// TwinCAT 3 PLC project IntelligenteWZM_PLCProject
// ProgramVersion: 3.1.4022.4
// libraries:
//   Tc2_Standard, * (Beckhoff Automation GmbH)
//   Tc2_System, * (Beckhoff Automation GmbH)
//   Tc3_Module, * (Beckhoff Automation GmbH)
//   VisuDialogs, * (System)
//   VisuSymbols,3.5.10.0,System
// project tree:
//   DUTs/ DW_TO_REAL.TcDUT
//   / GlobalTextList.TcGTLO (not stored), PlcTask.TcTTO, Visualization Manager.TcVMO (not stored)
//   GVLs/ GVarL.TcGVL
//   POUs/ ADAS_Kom.TcPOU, ANALOG_INPUT_EL3104.TcPOU, ANALOG_OUTPUT_EL4134.TcPOU (not stored), DATAMODULE.TcPOU (not stored), DATA_PREPARATION.TcPOU (not stored), DEFLECTION_CONTROL_FEED.TcPOU, DEFLECTION_CONTROL_POSITION.TcPOU (not stored), DP_CONFIG_IN_EL6731.TcPOU (not stored), DP_CONFIG_OUT_EL6731.TcPOU, ELLIP_FILTER.TcPOU (not stored), FORCE_SIGNALS.TcPOU, MAIN.TcPOU, MEAS_STIFFNESS_COLLISION.TcPOU (not stored), MEAS_STIFFNESS_PROCESS.TcPOU (not stored), Test.TcPOU (not stored), TOUCH_PROBE_LINE.TcPOU, VARIABLES.TcGVL (not stored), SENSOR_CONTROL_EL6751.TcPOU, SENSOR_SIGNALS_EL6751.TcPOU
//   VISUs/ Datamodule.TcVIS (not stored), PICTURES.TcIPO (not stored), VISUALISATION_DEFLEC_CONTROL.TcVIS, VISUALISATION_EMO2017.TcVIS, VISUALISATION_SENSOR_CONTROL.TcVIS, VISUALISATION_STIFFNESS_COLLISION.TcVIS, VISUALISATION_STIFFNESS_PROCESS.TcVIS (not stored)
// real-time tasks:
//   TASK PlcTask: cycle T#1ms, priority 20, ADS port 350
//   TASK Task 1: cycle T#10ms, priority 1, ADS port 301
// I/O:
//   DEVICE Device 2 (EtherCAT), AmsNetId 169.254.30.239.3.1
//     Term 1 (EK1100) [EK1100 EtherCAT Coupler (2A E-Bus)]
//       Term 2 (EL4134) [EL4134 4Ch. Ana. Output -10/+10V, 16bit]
//       Term 3 (EL3104) [EL3104 4Ch. Ana. Input +/-10V Diff.]
//       Term 4 (EL6731-0010) [EL6731-0010 PROFIBUS DP Slave]
//       Term 5 (EL6751) [EL6751 CANopen Master]
//       Term 6 (EL9512) [EL9512 Power supply terminal 12V]
//       Term 11 (EL9011) [EL9011 End Terminal]
//     Term 7 (EK1100) [EK1100 EtherCAT Coupler (2A E-Bus)]
//       Term 8 (EL3632) [EL3632 2Ch. IEPE Sensor]
//       Term 9 (EL3632) [EL3632 2Ch. IEPE Sensor]
//       Term 10 (EL3632) [EL3632 2Ch. IEPE Sensor]
//       Term 12 (EL9011) [EL9011 End Terminal]
//   DEVICE Device 1 (EL6731-0010), AmsNetId 169.254.30.239.2.1
//     PROFIBUS-Sinumerik (EL6731-0010) // Vendor: BECKHOFF Revision: Revision 2.00
//   DEVICE Device 3 (EL6751), AmsNetId 169.254.30.239.4.1
//     CAN-Sensors (CANopen Node)
// variable links:
//   IntelligenteWZM_PLCProject/IntelligenteWZM_PLCProject Instance <-> Device 1 (EL6731-0010)/PROFIBUS-Sinumerik (EL6731-0010)
//     PlcTask Inputs/VARIABLES.DP_MOSI_WORD_{1..4} <-> Module {5..8} (1 WORD Slave-In/Master-Out)/Inputs/1 WORD Slave-In/Master-Out_0_0  (4 links)
//     PlcTask Outputs/VARIABLES.DP_MISO_WORD_{1..4} <-> Module {1..4} (1 WORD Slave-Out/Master-In)/Outputs/1 WORD Slave-Out/Master-In_1_0  (4 links)
//   IntelligenteWZM_PLCProject/IntelligenteWZM_PLCProject Instance <-> Device 2 (EtherCAT)/Term 7 (EK1100)/Term 10 (EL3632)
//     PlcTask Inputs/VARIABLES.A_OVERSAMPLING_INPUT_5[0] <-> Ch1 Sample 0/Ch1 Value
//     PlcTask Inputs/VARIABLES.A_OVERSAMPLING_INPUT_5[1] <-> Ch1 Sample 1/Ch1 Value
//     PlcTask Inputs/VARIABLES.A_OVERSAMPLING_INPUT_5[2] <-> Ch1 Sample 2/Ch1 Value
//     PlcTask Inputs/VARIABLES.A_OVERSAMPLING_INPUT_5[3] <-> Ch1 Sample 3/Ch1 Value
//     PlcTask Inputs/VARIABLES.A_OVERSAMPLING_INPUT_5[4] <-> Ch1 Sample 4/Ch1 Value
//     PlcTask Inputs/VARIABLES.A_OVERSAMPLING_INPUT_5[5] <-> Ch1 Sample 5/Ch1 Value
//     PlcTask Inputs/VARIABLES.A_OVERSAMPLING_INPUT_5[6] <-> Ch1 Sample 6/Ch1 Value
//     PlcTask Inputs/VARIABLES.A_OVERSAMPLING_INPUT_5[7] <-> Ch1 Sample 7/Ch1 Value
//     PlcTask Inputs/VARIABLES.A_OVERSAMPLING_INPUT_5[8] <-> Ch1 Sample 8/Ch1 Value
//     PlcTask Inputs/VARIABLES.A_OVERSAMPLING_INPUT_5[9] <-> Ch1 Sample 9/Ch1 Value
//     PlcTask Inputs/VARIABLES.A_OVERSAMPLING_INPUT_6[0] <-> Ch2 Sample 0/Ch2 Value
//     PlcTask Inputs/VARIABLES.A_OVERSAMPLING_INPUT_6[1] <-> Ch2 Sample 1/Ch2 Value
//     PlcTask Inputs/VARIABLES.A_OVERSAMPLING_INPUT_6[2] <-> Ch2 Sample 2/Ch2 Value
//     PlcTask Inputs/VARIABLES.A_OVERSAMPLING_INPUT_6[3] <-> Ch2 Sample 3/Ch2 Value
//     PlcTask Inputs/VARIABLES.A_OVERSAMPLING_INPUT_6[4] <-> Ch2 Sample 4/Ch2 Value
//     PlcTask Inputs/VARIABLES.A_OVERSAMPLING_INPUT_6[5] <-> Ch2 Sample 5/Ch2 Value
//     PlcTask Inputs/VARIABLES.A_OVERSAMPLING_INPUT_6[6] <-> Ch2 Sample 6/Ch2 Value
//     PlcTask Inputs/VARIABLES.A_OVERSAMPLING_INPUT_6[7] <-> Ch2 Sample 7/Ch2 Value
//     PlcTask Inputs/VARIABLES.A_OVERSAMPLING_INPUT_6[8] <-> Ch2 Sample 8/Ch2 Value
//     PlcTask Inputs/VARIABLES.A_OVERSAMPLING_INPUT_6[9] <-> Ch2 Sample 9/Ch2 Value
//   IntelligenteWZM_PLCProject/IntelligenteWZM_PLCProject Instance <-> Device 2 (EtherCAT)/Term 7 (EK1100)/Term 8 (EL3632)
//     PlcTask Inputs/VARIABLES.A_OVERSAMPLING_INPUT_1[0] <-> Ch1 Sample 0/Ch1 Value
//     PlcTask Inputs/VARIABLES.A_OVERSAMPLING_INPUT_1[1] <-> Ch1 Sample 1/Ch1 Value
//     PlcTask Inputs/VARIABLES.A_OVERSAMPLING_INPUT_1[2] <-> Ch1 Sample 2/Ch1 Value
//     PlcTask Inputs/VARIABLES.A_OVERSAMPLING_INPUT_1[3] <-> Ch1 Sample 3/Ch1 Value
//     PlcTask Inputs/VARIABLES.A_OVERSAMPLING_INPUT_1[4] <-> Ch1 Sample 4/Ch1 Value
//     PlcTask Inputs/VARIABLES.A_OVERSAMPLING_INPUT_1[5] <-> Ch1 Sample 5/Ch1 Value
//     PlcTask Inputs/VARIABLES.A_OVERSAMPLING_INPUT_1[6] <-> Ch1 Sample 6/Ch1 Value
//     PlcTask Inputs/VARIABLES.A_OVERSAMPLING_INPUT_1[7] <-> Ch1 Sample 7/Ch1 Value
//     PlcTask Inputs/VARIABLES.A_OVERSAMPLING_INPUT_1[8] <-> Ch1 Sample 8/Ch1 Value
//     PlcTask Inputs/VARIABLES.A_OVERSAMPLING_INPUT_1[9] <-> Ch1 Sample 9/Ch1 Value
//     PlcTask Inputs/VARIABLES.A_OVERSAMPLING_INPUT_2[0] <-> Ch2 Sample 0/Ch2 Value
//     PlcTask Inputs/VARIABLES.A_OVERSAMPLING_INPUT_2[1] <-> Ch2 Sample 1/Ch2 Value
//     PlcTask Inputs/VARIABLES.A_OVERSAMPLING_INPUT_2[2] <-> Ch2 Sample 2/Ch2 Value
//     PlcTask Inputs/VARIABLES.A_OVERSAMPLING_INPUT_2[3] <-> Ch2 Sample 3/Ch2 Value
//     PlcTask Inputs/VARIABLES.A_OVERSAMPLING_INPUT_2[4] <-> Ch2 Sample 4/Ch2 Value
//     PlcTask Inputs/VARIABLES.A_OVERSAMPLING_INPUT_2[5] <-> Ch2 Sample 5/Ch2 Value
//     PlcTask Inputs/VARIABLES.A_OVERSAMPLING_INPUT_2[6] <-> Ch2 Sample 6/Ch2 Value
//     PlcTask Inputs/VARIABLES.A_OVERSAMPLING_INPUT_2[7] <-> Ch2 Sample 7/Ch2 Value
//     PlcTask Inputs/VARIABLES.A_OVERSAMPLING_INPUT_2[8] <-> Ch2 Sample 8/Ch2 Value
//     PlcTask Inputs/VARIABLES.A_OVERSAMPLING_INPUT_2[9] <-> Ch2 Sample 9/Ch2 Value
//   IntelligenteWZM_PLCProject/IntelligenteWZM_PLCProject Instance <-> Device 2 (EtherCAT)/Term 7 (EK1100)/Term 9 (EL3632)
//     PlcTask Inputs/VARIABLES.A_OVERSAMPLING_INPUT_3[0] <-> Ch1 Sample 0/Ch1 Value
//     PlcTask Inputs/VARIABLES.A_OVERSAMPLING_INPUT_3[1] <-> Ch1 Sample 1/Ch1 Value
//     PlcTask Inputs/VARIABLES.A_OVERSAMPLING_INPUT_3[2] <-> Ch1 Sample 2/Ch1 Value
//     PlcTask Inputs/VARIABLES.A_OVERSAMPLING_INPUT_3[3] <-> Ch1 Sample 3/Ch1 Value
//     PlcTask Inputs/VARIABLES.A_OVERSAMPLING_INPUT_3[4] <-> Ch1 Sample 4/Ch1 Value
//     PlcTask Inputs/VARIABLES.A_OVERSAMPLING_INPUT_3[5] <-> Ch1 Sample 5/Ch1 Value
//     PlcTask Inputs/VARIABLES.A_OVERSAMPLING_INPUT_3[6] <-> Ch1 Sample 6/Ch1 Value
//     PlcTask Inputs/VARIABLES.A_OVERSAMPLING_INPUT_3[7] <-> Ch1 Sample 7/Ch1 Value
//     PlcTask Inputs/VARIABLES.A_OVERSAMPLING_INPUT_3[8] <-> Ch1 Sample 8/Ch1 Value
//     PlcTask Inputs/VARIABLES.A_OVERSAMPLING_INPUT_3[9] <-> Ch1 Sample 9/Ch1 Value
//     PlcTask Inputs/VARIABLES.A_OVERSAMPLING_INPUT_4[0] <-> Ch2 Sample 0/Ch2 Value
//     PlcTask Inputs/VARIABLES.A_OVERSAMPLING_INPUT_4[1] <-> Ch2 Sample 1/Ch2 Value
//     PlcTask Inputs/VARIABLES.A_OVERSAMPLING_INPUT_4[2] <-> Ch2 Sample 2/Ch2 Value
//     PlcTask Inputs/VARIABLES.A_OVERSAMPLING_INPUT_4[3] <-> Ch2 Sample 3/Ch2 Value
//     PlcTask Inputs/VARIABLES.A_OVERSAMPLING_INPUT_4[4] <-> Ch2 Sample 4/Ch2 Value
//     PlcTask Inputs/VARIABLES.A_OVERSAMPLING_INPUT_4[5] <-> Ch2 Sample 5/Ch2 Value
//     PlcTask Inputs/VARIABLES.A_OVERSAMPLING_INPUT_4[6] <-> Ch2 Sample 6/Ch2 Value
//     PlcTask Inputs/VARIABLES.A_OVERSAMPLING_INPUT_4[7] <-> Ch2 Sample 7/Ch2 Value
//     PlcTask Inputs/VARIABLES.A_OVERSAMPLING_INPUT_4[8] <-> Ch2 Sample 8/Ch2 Value
//     PlcTask Inputs/VARIABLES.A_OVERSAMPLING_INPUT_4[9] <-> Ch2 Sample 9/Ch2 Value
//   IntelligenteWZM_PLCProject/IntelligenteWZM_PLCProject Instance <-> Device 3 (EL6751)/CAN-Sensors (CANopen Node)
//     PlcTask Inputs/VARIABLES.CAN_SENSOR_{1..10} <-> Sensor ID {1..10}/Inputs/CAN_IN_MESSAGE_D{1..10}  (10 links)
//     PlcTask Outputs/VARIABLES.CAN_HUB <-> HUB Control ID 0/Outputs/CAN_OUT_MESSAGE_CONTROL

CONFIGURATION IntelligenteWZM_PLCProject
    RESOURCE PLC ON TwinCAT3
        TASK PlcTask(INTERVAL := T#1ms, PRIORITY := 20);
        PROGRAM MAIN WITH PlcTask : MAIN;
    END_RESOURCE
END_CONFIGURATION

// ---- DUTs/DW_TO_REAL.TcDUT
TYPE DW_TO_REAL :
UNION
	IntAsWord : ARRAY[0..1] OF WORD;
	IntAsReal: REAL;
END_UNION
END_TYPE

// ---- GVLs/GVarL.TcGVL
VAR_GLOBAL
	///ADAS 
	iSignalID: ARRAY[0..20] OF BYTE;
	iAchseID: ARRAY[0..20] OF BYTE;
	iComCylce: BYTE := 20;
	iMode: INT := 10;
	iTracks: UINT;
	///Position x
	X_Machine_CS AT %Q*: LREAL;
	///Position y
	Y_Machine_CS AT %Q*: LREAL;
	///Position z
	Z_Machine_CS AT %Q*: LREAL;
	///Position c
	C_Machine_CS AT %Q*: LREAL;
	///Position b
	B_Machine_CS AT %Q*: LREAL;
	///Soll-Position x
	X_Machine_CS_soll AT %Q*: LREAL;
	///Geschwindigkeit x
	X_V_Machine_CS AT %Q*: LREAL;
	///Geschwindigkeit y
	Y_V_Machine_CS AT %Q*: LREAL;
	///Geschwindigkeit z
	Z_V_Machine_CS AT %Q*: LREAL;
	///Geschwindigkeit c
	C_V_Machine_CS AT %Q*: LREAL;
	///Geschwindigkeit b
	B_V_Machine_CS AT %Q*: LREAL;
	///Drehzahl n
	n_Spindle AT %Q*: LREAL;
	///Beschleunigung x
	X_a_Machine_CS AT %Q*: LREAL;
	///Beschleunigung y
	Y_a_Machine_CS AT %Q*: LREAL;
	///Beschleunigung z
	Z_a_Machine_CS AT %Q*: LREAL;
	///Beschleunigung c
	C_a_Machine_CS AT %Q*: LREAL;
	///Beschleunigung b
	B_a_Machine_CS AT %Q*: LREAL;
	///Strom x
	X_I AT %Q*: LREAL;
	///Strom y
	Y_I AT %Q*: LREAL;
	///Strom z
	Z_I AT %Q*: LREAL;
	///Strom c
	C_I AT %Q*: LREAL;
	///Strom b
	B_I AT %Q*: LREAL;
	///Strom Spindel
	n_I AT %Q*: LREAL;
	Data: uCCDatagram;
	///CCDataStreamSetupOUT 	 		:sCCDataStreamSetup;
	CCDataStreamSetupOUT AT %Q*: sCCDataStreamSetup;
	bGO: BOOL;

	XSynVar: LREAL;
END_VAR

VAR_GLOBAL CONSTANT
	///ADAS
	gVar_NumberOfAdasTracks: INT := 30;
END_VAR

// ---- POUs/MAIN.TcPOU
PROGRAM MAIN
VAR_INPUT
//ADAS
	ADAS_in		AT %I* 	: ARRAY[0..63] OF WORD; //ADAS_Rohdaten
END_VAR


IF FORCE_RESET=1 THEN
	RESULT[0]:=0;
	PTS_MEASUREMENT_HISTOGRAM_2[2]:=0;
	RESULT[1]:=0;
END_IF

IF VarTest = TRUE THEN
	VarTest := FALSE;
END_IF

IF VarTest = FALSE THEN
	VarTest := TRUE;
END_IF

ANALOG_INPUT_EL3104();
//ANALOG_OUTPUT_EL4134();
DP_CONFIG_IN_EL6731();
SENSOR_CONTROL_EL6751();
SENSOR_SIGNALS_EL6751();
FORCE_SIGNALS();
//Test();
DATAMODULE();

MEAS_STIFFNESS_COLLISION();
MEAS_STIFFNESS_PROCESS();
DEFLECTION_CONTROL_FEED();
DEFLECTION_CONTROL_POSITION();
TOUCH_PROBE_LINE();
DP_CONFIG_OUT_EL6731();


//ADAS Daten
	//x-Achse (soll alles stimmen)
X_Machine_CS 		:= DINT_TO_LREAL(ADAS_Kom.adasData[1])	/ 10000; //Umrechnung in: mm -> /10000 (10000 inkremente sind 1mm)
X_Machine_CS_soll 	:= DINT_TO_LREAL(ADAS_Kom.adasData[27])	/ 10000; //Umrechnung in: mm -> /10000 (10000 inkremente sind 1mm)
X_V_Machine_CS 		:= DINT_TO_LREAL(ADAS_Kom.adasData[6])	/ 10000; //Umrechnung in: mm/s-> /10000
X_a_Machine_CS 		:= DINT_TO_LREAL(ADAS_Kom.adasData[12])	/ 10000; //Umrechnung in: mm/s²-> /10000
X_I					:= DINT_TO_LREAL(ADAS_Kom.adasData[18])	/ 1000;  //Umrechnung in: A -> /1000

	//y-Achse  (soll alles stimmen)
Y_Machine_CS 		:= DINT_TO_LREAL(ADAS_Kom.adasData[2]) 	/ 10000; //Umrechnung in: mm -> /10000
Y_V_Machine_CS 		:= DINT_TO_LREAL(ADAS_Kom.adasData[7]) 	/ 10000; //Umrechnung in: mm/s-> /10000
Y_a_Machine_CS 		:= DINT_TO_LREAL(ADAS_Kom.adasData[13])	/ 10000; //Umrechnung in: mm/s²-> /10000
Y_I					:= DINT_TO_LREAL(ADAS_Kom.adasData[19])	/ 1000;  //Umrechnung in: A -> /1000
	//z-Achse (soll alles stimmen)
Z_Machine_CS 		:= DINT_TO_LREAL(ADAS_Kom.adasData[3]) 	/ 10000; //Umrechnung in: mm -> /10000
Z_V_Machine_CS 		:= DINT_TO_LREAL(ADAS_Kom.adasData[8]) 	/ 10000; //Umrechnung in: mm/s-> /10000
Z_a_Machine_CS 		:= DINT_TO_LREAL(ADAS_Kom.adasData[14])	/ 10000; //Umrechnung in: mm/s²-> /10000
Z_I					:= DINT_TO_LREAL(ADAS_Kom.adasData[20])	/ 1000;  //Umrechnung in: A -> /1000
	//C-Achse (soll alles stimmen)
C_Machine_CS 		:= DINT_TO_LREAL(ADAS_Kom.adasData[4]) 	/ 10000; //Umrechnung in: mm -> /10000
C_V_Machine_CS 		:= DINT_TO_LREAL(ADAS_Kom.adasData[9]) 	/ 10000; //Umrechnung in: mm/s-> /10000
C_a_Machine_CS 		:= DINT_TO_LREAL(ADAS_Kom.adasData[15])	/ 10000; //Umrechnung in: mm/s²-> /10000
C_I 				:= DINT_TO_LREAL(ADAS_Kom.adasData[21])	/ 1000;  //Umrechnung in: A -> /1000
	//B-Achse (B_Machine_CS wid von Spinel beschrieben)
B_Machine_CS		:= DINT_TO_LREAL(ADAS_Kom.adasData[24]) / 10000; //Umrechnung in: mm -> /10000 //b
B_V_Machine_CS 		:= DINT_TO_LREAL(ADAS_Kom.adasData[10]) / 10000; //Umrechnung in: mm/s-> /10000
B_a_Machine_CS 		:= DINT_TO_LREAL(ADAS_Kom.adasData[16]) / 10000; //Umrechnung in: mm/s²-> /10000
B_I 				:= DINT_TO_LREAL(ADAS_Kom.adasData[22]) / 1000;  //Umrechnung in: A -> /1000
	//Spindel
n_Spindle 			:= (DINT_TO_LREAL(ADAS_Kom.adasData[5])/360)*60/10000 ; //kommt in milli°/s Umrechnung in: 1/min-> *0,166667
n_I 				:= DINT_TO_LREAL(ADAS_Kom.adasData[25])/1000; //Umrechnung in: A -> /1000

END_PROGRAM

// ---- POUs/ANALOG_INPUT_EL3104.TcPOU
PROGRAM ANALOG_INPUT_EL3104
VAR
END_VAR


A_SIGNAL_1 := INT_TO_REAL(A_INPUT_1)*A_GAIN_1*10/ 32767;
A_SIGNAL_2 := INT_TO_REAL(A_INPUT_2)*A_GAIN_2*10/ 32767;
A_SIGNAL_3 := INT_TO_REAL(A_INPUT_3)*A_GAIN_3*10/ 32767;
A_SIGNAL_4 := INT_TO_REAL(A_INPUT_4)*A_GAIN_4*10/ 32767;

END_PROGRAM

// ---- POUs/SENSOR_CONTROL_EL6751.TcPOU
PROGRAM SENSOR_CONTROL_EL6751
VAR
	Samp: WORD:=0;	
	FigArray: ARRAY [0..7] OF USINT :=[0, 0, 0, 0, 0, 0, 0, 0];
	Previous: USINT:=16#0;
END_VAR

HUB_STATE:=FALSE; 

IF CAN_TRIGGER_STATE=1 AND M_PER_FRAME=1 THEN
	CAN_CONTROL_FRAME:=FigArray;
	IF samp>K_Trigger THEN			// Can occurs by changing M_PER_FRAME from 2,3 or 4 to 1 
		samp:=0;
	END_IF
	Samp:=Samp+1;
	IF Samp=K_Trigger THEN
		CAN_CONTROL_FRAME[0]:=16#3;
		CAN_CONTROL_FRAME[2]:=16#1;
		CAN_CONTROL_FRAME[4]:=N_SAMPLES_PER_M;
		CASE Previous OF
			16#0: 	CAN_CONTROL_FRAME[3]:=16#0;
					Previous:=16#1;
			16#1: 	CAN_CONTROL_FRAME[3]:=16#1;
					Previous:=16#0;
		END_CASE
		SIGNAL_SYNCH:=1;
		Samp:=0;
		CAN_HUB:=CAN_CONTROL_FRAME;	
	END_IF	
	HUB_STATE:=TRUE;
END_IF



IF CAN_TRIGGER_STATE=1 AND M_PER_FRAME=2 THEN
	CAN_CONTROL_FRAME:=FigArray;
	Samp:=Samp+1;
	IF Samp=K_Trigger OR Samp=(2*K_Trigger) THEN
		CAN_CONTROL_FRAME[0]:=16#3;
		CAN_CONTROL_FRAME[2]:=16#2;
		CAN_CONTROL_FRAME[4]:=N_SAMPLES_PER_M;
		IF Samp=K_Trigger THEN
			CAN_CONTROL_FRAME[3]:=16#1;
			SIGNAL_SYNCH:=1;
		END_IF
		IF Samp=(2*K_Trigger) THEN
			CAN_CONTROL_FRAME[3]:=16#2;
			SIGNAL_SYNCH:=2;
			Samp:=0;
		END_IF
		CAN_HUB:=CAN_CONTROL_FRAME;	
	END_IF
	HUB_STATE:=TRUE;
END_IF



IF CAN_TRIGGER_STATE=1 AND M_PER_FRAME=3 THEN
	CAN_CONTROL_FRAME:=FigArray;
	Samp:=Samp+1;
	IF Samp=K_Trigger OR Samp=(2*K_Trigger) OR Samp=(3*K_Trigger) THEN
		CAN_CONTROL_FRAME[0]:=16#3;
		CAN_CONTROL_FRAME[2]:=16#3;
		CAN_CONTROL_FRAME[4]:=N_SAMPLES_PER_M;
		IF Samp=K_Trigger THEN
			CAN_CONTROL_FRAME[3]:=16#1;
			SIGNAL_SYNCH:=1;
		END_IF
		IF Samp=(2*K_Trigger) THEN
			CAN_CONTROL_FRAME[3]:=16#2;
			SIGNAL_SYNCH:=2;
		END_IF
		IF Samp=(3*K_Trigger) THEN
			CAN_CONTROL_FRAME[3]:=16#3;
			SIGNAL_SYNCH:=3;
			Samp:=0;
		END_IF
		CAN_HUB:=CAN_CONTROL_FRAME;	
	END_IF
	HUB_STATE:=TRUE;
END_IF


IF CAN_TRIGGER_STATE=1 AND M_PER_FRAME=4 THEN
	CAN_CONTROL_FRAME:=FigArray;
	Samp:=Samp+1;
	IF Samp=K_Trigger OR Samp=(2*K_Trigger) OR Samp=(3*K_Trigger) OR Samp=(4*K_Trigger)  THEN
		CAN_CONTROL_FRAME[0]:=16#3;
		CAN_CONTROL_FRAME[2]:=16#4;
		CAN_CONTROL_FRAME[4]:=N_SAMPLES_PER_M;
		IF Samp=K_Trigger THEN
			CAN_CONTROL_FRAME[3]:=16#1;
			SIGNAL_SYNCH:=1;
		END_IF
		IF Samp=(2*K_Trigger) THEN
			CAN_CONTROL_FRAME[3]:=16#2;
			SIGNAL_SYNCH:=2;
		END_IF
		IF Samp=(3*K_Trigger) THEN
			CAN_CONTROL_FRAME[3]:=16#3;
			SIGNAL_SYNCH:=3;
		END_IF
		IF Samp=(4*K_Trigger) THEN
			CAN_CONTROL_FRAME[3]:=16#4;
			SIGNAL_SYNCH:=4;
			Samp:=0;
		END_IF
		CAN_HUB:=CAN_CONTROL_FRAME;		
	END_IF
	HUB_STATE:=TRUE;
END_IF

IF CAN_CONTROL_STATE=0 THEN
	CAN_CONTROL_FRAME:=FigArray;
	CAN_CONTROL_FRAME[0]:=16#0;
	CAN_HUB:=CAN_CONTROL_FRAME;
	CAN_CONTROL_STATE:=11;
	HUB_STATE:=TRUE;
END_IF

IF CAN_CONTROL_STATE=1 THEN
	CAN_CONTROL_FRAME:=FigArray;
	CAN_CONTROL_FRAME[0]:=16#1;
	CAN_HUB:=CAN_CONTROL_FRAME;
	CAN_CONTROL_STATE:=11;
	HUB_STATE:=TRUE;
END_IF

IF CAN_CONTROL_STATE=2 THEN
	CAN_CONTROL_FRAME:=FigArray;
	CAN_CONTROL_FRAME[0]:=16#2;
	CAN_HUB:=CAN_CONTROL_FRAME;
	CAN_CONTROL_STATE:=11;
	HUB_STATE:=TRUE;
END_IF

IF CAN_CONTROL_STATE=3 THEN
	CAN_CONTROL_FRAME:=CAN_PARAMETER_FRAME;
	CAN_HUB:=CAN_CONTROL_FRAME;
	CAN_CONTROL_STATE:=11;
	CAN_PARAMETER_FRAME:=FigArray;
	HUB_STATE:=TRUE;
END_IF

END_PROGRAM

// ---- POUs/SENSOR_SIGNALS_EL6751.TcPOU
PROGRAM SENSOR_SIGNALS_EL6751
VAR
	FILTER_S1:ELLIP_FILTER;
	FILTER_S2:ELLIP_FILTER;
	FILTER_S3:ELLIP_FILTER;
	FILTER_S4:ELLIP_FILTER;
	FILTER_S5:ELLIP_FILTER;
	FILTER_S6:ELLIP_FILTER;
	FILTER_S7:ELLIP_FILTER;
	FILTER_S8:ELLIP_FILTER;
	FILTER_S9:ELLIP_FILTER;
	FILTER_S10:ELLIP_FILTER;
	
	
	Calc_Dev: ARRAY[1..3,1..10] OF LREAL:=[0, 0, 0, 0, 0, 0, 0, 0, 0, 0, 0, 0, 0, 0, 0, 0, 0, 0, 0, 0, 0, 0, 0, 0, 0, 0, 0, 0, 0, 0 ];
	k: WORD;
	Signal_5: WORD:=0;
	Signal_1: WORD:=0;
	Mem_Signal_1: ARRAY[1..10] OF WORD:=[0,0,0,0,0,0,0,0,0,0];
	N_Mem_Sig_1: ARRAY[1..10] OF WORD:=[0,0,0,0,0,0,0,0,0,0];
	N_Dev: WORD:=500;
	
END_VAR

//SENSOR 1
SIGNAL_SENSOR_1[1]:=SHL(CAN_SENSOR_1[0],8)+CAN_SENSOR_1[1];
SIGNAL_SENSOR_1[2]:=SHL(CAN_SENSOR_1[2],8)+CAN_SENSOR_1[3];
SIGNAL_SENSOR_1[3]:=SHL(CAN_SENSOR_1[4],8)+CAN_SENSOR_1[5];
SIGNAL_SENSOR_1[4]:=SHL(CAN_SENSOR_1[6],8)+CAN_SENSOR_1[7];
CASE SIGNAL_SYNCH OF
	1: SIGNAL_SENSOR_1[5]:=SIGNAL_SENSOR_1[1];
	2: SIGNAL_SENSOR_1[5]:=SIGNAL_SENSOR_1[2];
	3: SIGNAL_SENSOR_1[5]:=SIGNAL_SENSOR_1[3];
	4: SIGNAL_SENSOR_1[5]:=SIGNAL_SENSOR_1[4];
END_CASE

//SENSOR 2
SIGNAL_SENSOR_2[1]:=SHL(CAN_SENSOR_2[0],8)+CAN_SENSOR_2[1];
SIGNAL_SENSOR_2[2]:=SHL(CAN_SENSOR_2[2],8)+CAN_SENSOR_2[3];
SIGNAL_SENSOR_2[3]:=SHL(CAN_SENSOR_2[4],8)+CAN_SENSOR_2[5];
SIGNAL_SENSOR_2[4]:=SHL(CAN_SENSOR_2[6],8)+CAN_SENSOR_2[7];
CASE SIGNAL_SYNCH OF
	1: SIGNAL_SENSOR_2[5]:=SIGNAL_SENSOR_2[1];
	2: SIGNAL_SENSOR_2[5]:=SIGNAL_SENSOR_2[2];
	3: SIGNAL_SENSOR_2[5]:=SIGNAL_SENSOR_2[3];
	4: SIGNAL_SENSOR_2[5]:=SIGNAL_SENSOR_2[4];
END_CASE

//SENSOR 3
SIGNAL_SENSOR_3[1]:=SHL(CAN_SENSOR_3[0],8)+CAN_SENSOR_3[1];
SIGNAL_SENSOR_3[2]:=SHL(CAN_SENSOR_3[2],8)+CAN_SENSOR_3[3];
SIGNAL_SENSOR_3[3]:=SHL(CAN_SENSOR_3[4],8)+CAN_SENSOR_3[5];
SIGNAL_SENSOR_3[4]:=SHL(CAN_SENSOR_3[6],8)+CAN_SENSOR_3[7];
CASE SIGNAL_SYNCH OF
	1: SIGNAL_SENSOR_3[5]:=SIGNAL_SENSOR_3[1];
	2: SIGNAL_SENSOR_3[5]:=SIGNAL_SENSOR_3[2];
	3: SIGNAL_SENSOR_3[5]:=SIGNAL_SENSOR_3[3];
	4: SIGNAL_SENSOR_3[5]:=SIGNAL_SENSOR_3[4];
END_CASE

//SENSOR 4
SIGNAL_SENSOR_4[1]:=SHL(CAN_SENSOR_4[0],8)+CAN_SENSOR_4[1];
SIGNAL_SENSOR_4[2]:=SHL(CAN_SENSOR_4[2],8)+CAN_SENSOR_4[3];
SIGNAL_SENSOR_4[3]:=SHL(CAN_SENSOR_4[4],8)+CAN_SENSOR_4[5];
SIGNAL_SENSOR_4[4]:=SHL(CAN_SENSOR_4[6],8)+CAN_SENSOR_4[7];
CASE SIGNAL_SYNCH OF
	1: SIGNAL_SENSOR_4[5]:=SIGNAL_SENSOR_4[1];
	2: SIGNAL_SENSOR_4[5]:=SIGNAL_SENSOR_4[2];
	3: SIGNAL_SENSOR_4[5]:=SIGNAL_SENSOR_4[3];
	4: SIGNAL_SENSOR_4[5]:=SIGNAL_SENSOR_4[4];
END_CASE

//SENSOR 5
SIGNAL_SENSOR_5[1]:=SHL(CAN_SENSOR_5[0],8)+CAN_SENSOR_5[1];
SIGNAL_SENSOR_5[2]:=SHL(CAN_SENSOR_5[2],8)+CAN_SENSOR_5[3];
SIGNAL_SENSOR_5[3]:=SHL(CAN_SENSOR_5[4],8)+CAN_SENSOR_5[5];
SIGNAL_SENSOR_5[4]:=SHL(CAN_SENSOR_5[6],8)+CAN_SENSOR_5[7];
CASE SIGNAL_SYNCH OF
	1: SIGNAL_SENSOR_5[5]:=SIGNAL_SENSOR_5[1];
	2: SIGNAL_SENSOR_5[5]:=SIGNAL_SENSOR_5[2];
	3: SIGNAL_SENSOR_5[5]:=SIGNAL_SENSOR_5[3];
	4: SIGNAL_SENSOR_5[5]:=SIGNAL_SENSOR_5[4];
END_CASE

//SENSOR 6
SIGNAL_SENSOR_6[1]:=SHL(CAN_SENSOR_6[0],8)+CAN_SENSOR_6[1];
SIGNAL_SENSOR_6[2]:=SHL(CAN_SENSOR_6[2],8)+CAN_SENSOR_6[3];
SIGNAL_SENSOR_6[3]:=SHL(CAN_SENSOR_6[4],8)+CAN_SENSOR_6[5];
SIGNAL_SENSOR_6[4]:=SHL(CAN_SENSOR_6[6],8)+CAN_SENSOR_6[7];
CASE SIGNAL_SYNCH OF
	1: SIGNAL_SENSOR_6[5]:=SIGNAL_SENSOR_6[1];
	2: SIGNAL_SENSOR_6[5]:=SIGNAL_SENSOR_6[2];
	3: SIGNAL_SENSOR_6[5]:=SIGNAL_SENSOR_6[3];
	4: SIGNAL_SENSOR_6[5]:=SIGNAL_SENSOR_6[4];
END_CASE

//SENSOR 7
SIGNAL_SENSOR_7[1]:=SHL(CAN_SENSOR_7[0],8)+CAN_SENSOR_7[1];
SIGNAL_SENSOR_7[2]:=SHL(CAN_SENSOR_7[2],8)+CAN_SENSOR_7[3];
SIGNAL_SENSOR_7[3]:=SHL(CAN_SENSOR_7[4],8)+CAN_SENSOR_7[5];
SIGNAL_SENSOR_7[4]:=SHL(CAN_SENSOR_7[6],8)+CAN_SENSOR_7[7];
CASE SIGNAL_SYNCH OF
	1: SIGNAL_SENSOR_7[5]:=SIGNAL_SENSOR_7[1];
	2: SIGNAL_SENSOR_7[5]:=SIGNAL_SENSOR_7[2];
	3: SIGNAL_SENSOR_7[5]:=SIGNAL_SENSOR_7[3];
	4: SIGNAL_SENSOR_7[5]:=SIGNAL_SENSOR_7[4];
END_CASE

//SENSOR 8
SIGNAL_SENSOR_8[1]:=SHL(CAN_SENSOR_8[0],8)+CAN_SENSOR_8[1];
SIGNAL_SENSOR_8[2]:=SHL(CAN_SENSOR_8[2],8)+CAN_SENSOR_8[3];
SIGNAL_SENSOR_8[3]:=SHL(CAN_SENSOR_8[4],8)+CAN_SENSOR_8[5];
SIGNAL_SENSOR_8[4]:=SHL(CAN_SENSOR_8[6],8)+CAN_SENSOR_8[7];
CASE SIGNAL_SYNCH OF
	1: SIGNAL_SENSOR_8[5]:=SIGNAL_SENSOR_8[1];
	2: SIGNAL_SENSOR_8[5]:=SIGNAL_SENSOR_8[2];
	3: SIGNAL_SENSOR_8[5]:=SIGNAL_SENSOR_8[3];
	4: SIGNAL_SENSOR_8[5]:=SIGNAL_SENSOR_8[4];
END_CASE

//SENSOR 9
SIGNAL_SENSOR_9[1]:=SHL(CAN_SENSOR_9[0],8)+CAN_SENSOR_9[1];
SIGNAL_SENSOR_9[2]:=SHL(CAN_SENSOR_9[2],8)+CAN_SENSOR_9[3];
SIGNAL_SENSOR_9[3]:=SHL(CAN_SENSOR_9[4],8)+CAN_SENSOR_9[5];
SIGNAL_SENSOR_9[4]:=SHL(CAN_SENSOR_9[6],8)+CAN_SENSOR_9[7];
CASE SIGNAL_SYNCH OF
	1: SIGNAL_SENSOR_9[5]:=SIGNAL_SENSOR_9[1];
	2: SIGNAL_SENSOR_9[5]:=SIGNAL_SENSOR_9[2];
	3: SIGNAL_SENSOR_9[5]:=SIGNAL_SENSOR_9[3];
	4: SIGNAL_SENSOR_9[5]:=SIGNAL_SENSOR_9[4];
END_CASE

//SENSOR 10
SIGNAL_SENSOR_10[1]:=SHL(CAN_SENSOR_10[0],8)+CAN_SENSOR_10[1];
SIGNAL_SENSOR_10[2]:=SHL(CAN_SENSOR_10[2],8)+CAN_SENSOR_10[3];
SIGNAL_SENSOR_10[3]:=SHL(CAN_SENSOR_10[4],8)+CAN_SENSOR_10[5];
SIGNAL_SENSOR_10[4]:=SHL(CAN_SENSOR_10[6],8)+CAN_SENSOR_10[7];
CASE SIGNAL_SYNCH OF
	1: SIGNAL_SENSOR_10[5]:=SIGNAL_SENSOR_10[1];
	2: SIGNAL_SENSOR_10[5]:=SIGNAL_SENSOR_10[2];
	3: SIGNAL_SENSOR_10[5]:=SIGNAL_SENSOR_10[3];
	4: SIGNAL_SENSOR_10[5]:=SIGNAL_SENSOR_10[4];
END_CASE

// SIGNAL FILTERING
FILTER_S1(ssMethodType:=1 , IN:= SIGNAL_SENSOR_1[5], OUT=> SIGNAL_SENSOR_1_FLT);
FILTER_S2(ssMethodType:=1 , IN:= SIGNAL_SENSOR_2[5], OUT=> SIGNAL_SENSOR_2_FLT);
FILTER_S3(ssMethodType:=1 , IN:= SIGNAL_SENSOR_3[5], OUT=> SIGNAL_SENSOR_3_FLT);
FILTER_S4(ssMethodType:=1 , IN:= SIGNAL_SENSOR_4[5], OUT=> SIGNAL_SENSOR_4_FLT);
FILTER_S5(ssMethodType:=1 , IN:= SIGNAL_SENSOR_5[5], OUT=> SIGNAL_SENSOR_5_FLT);
FILTER_S6(ssMethodType:=1 , IN:= SIGNAL_SENSOR_6[5], OUT=> SIGNAL_SENSOR_6_FLT);
FILTER_S7(ssMethodType:=1 , IN:= SIGNAL_SENSOR_7[5], OUT=> SIGNAL_SENSOR_7_FLT);
FILTER_S8(ssMethodType:=1 , IN:= SIGNAL_SENSOR_8[5], OUT=> SIGNAL_SENSOR_8_FLT);
FILTER_S9(ssMethodType:=1 , IN:= SIGNAL_SENSOR_9[5], OUT=> SIGNAL_SENSOR_9_FLT);
FILTER_S10(ssMethodType:=1 , IN:= SIGNAL_SENSOR_10[5], OUT=> SIGNAL_SENSOR_10_FLT);

// SIGNAL DEVIATION AND SIGNAL STATE
FOR k:=1 TO 10 BY 1 DO
	Calc_Dev[1,k]:=Calc_Dev[1,k]+1;
	CASE k OF
		1: 	Signal_5:=SIGNAL_SENSOR_1[5];
			Signal_1:=SIGNAL_SENSOR_1[1];
		2: 	Signal_5:=SIGNAL_SENSOR_2[5];
			Signal_1:=SIGNAL_SENSOR_2[1];
		3: 	Signal_5:=SIGNAL_SENSOR_3[5];
			Signal_1:=SIGNAL_SENSOR_3[1];
		4: 	Signal_5:=SIGNAL_SENSOR_4[5];
			Signal_1:=SIGNAL_SENSOR_4[1];
		5: 	Signal_5:=SIGNAL_SENSOR_5[5];
			Signal_1:=SIGNAL_SENSOR_5[1];
		6: 	Signal_5:=SIGNAL_SENSOR_6[5];
			Signal_1:=SIGNAL_SENSOR_6[1];
		7: 	Signal_5:=SIGNAL_SENSOR_7[5];
			Signal_1:=SIGNAL_SENSOR_7[1];
		8: 	Signal_5:=SIGNAL_SENSOR_8[5];
			Signal_1:=SIGNAL_SENSOR_8[1];
		9: 	Signal_5:=SIGNAL_SENSOR_9[5];
			Signal_1:=SIGNAL_SENSOR_9[1];
		10: Signal_5:=SIGNAL_SENSOR_10[5];
			Signal_1:=SIGNAL_SENSOR_10[1];	
	END_CASE
	
	IF Calc_Dev[1,k]<N_Dev THEN
		Calc_Dev[2,k]:=Calc_Dev[2,k]+EXPT(WORD_TO_LREAL(Signal_5),2)/(N_Dev-1);
		Calc_Dev[3,k]:=Calc_Dev[3,k]+WORD_TO_LREAL(Signal_5);
	END_IF
	
	IF Calc_Dev[1,k]=N_Dev THEN
		IF Calc_Dev[2,k]-(EXPT(Calc_Dev[3,k],2)/EXPT((N_Dev-1),2))>=0 THEN
			SIGNAL_DEVIATION[k]:=LREAL_TO_WORD(3*SQRT(Calc_Dev[2,k]-(EXPT(Calc_Dev[3,k],2)/EXPT((N_Dev-1),2))));
			Calc_Dev[1,k]:=0;
			Calc_Dev[2,k]:=0;
			Calc_Dev[3,k]:=0;
			ELSE
				Calc_Dev[1,k]:=0;
				Calc_Dev[2,k]:=0;
				Calc_Dev[3,k]:=0;
				SIGNAL_DEVIATION[k]:=0;
		END_IF
	END_IF
	
	IF Signal_1<>Mem_Signal_1[k] THEN
		N_Mem_Sig_1[k]:=0;
		Mem_Signal_1[k]:=Signal_1;
		ELSE
		N_Mem_Sig_1[k]:=N_Mem_Sig_1[k]+1;
		Mem_Signal_1[k]:=Signal_1;
	END_IF
	
	IF N_Mem_Sig_1[k]< N_Dev THEN
		SENSOR_STATE[k]:=1;
		ELSE
			SENSOR_STATE[k]:=0;	
			SIGNAL_DEVIATION[k]:=0;	
	END_IF
	
END_FOR

END_PROGRAM

// ---- POUs/FORCE_SIGNALS.TcPOU
PROGRAM FORCE_SIGNALS
VAR
	RESET_FORCE_VAL: ARRAY[1..3] OF REAL := [0,0,0];
	FORCE_ROW: ARRAY[1..3] OF REAL;
	FORCE_SUM: ARRAY[1..3] OF REAL:= [0,0,0];
	INK: INT:=0;
	
	FILTER_FX:ELLIP_FILTER;
	FILTER_FY:ELLIP_FILTER;
	FILTER_FZ:ELLIP_FILTER;
	
	
END_VAR

FORCE_ROW[1]:=(FC_MATRIX_X[1]*SIGNAL_SENSOR_1[1]+FC_MATRIX_X[2]*SIGNAL_SENSOR_2[1]+FC_MATRIX_X[3]*SIGNAL_SENSOR_3[1]+FC_MATRIX_X[4]*SIGNAL_SENSOR_4[1]+FC_MATRIX_X[5]*SIGNAL_SENSOR_5[1]+FC_MATRIX_X[6]*SIGNAL_SENSOR_6[1]+FC_MATRIX_X[7]*SIGNAL_SENSOR_7[1]+FC_MATRIX_X[8]*SIGNAL_SENSOR_8[1]+FC_MATRIX_X[9]*SIGNAL_SENSOR_9[1]+FC_MATRIX_X[10]*SIGNAL_SENSOR_10[1]);
FORCE_ROW[2]:=(FC_MATRIX_Y[1]*SIGNAL_SENSOR_1[1]+FC_MATRIX_Y[2]*SIGNAL_SENSOR_2[1]+FC_MATRIX_Y[3]*SIGNAL_SENSOR_3[1]+FC_MATRIX_Y[4]*SIGNAL_SENSOR_4[1]+FC_MATRIX_Y[5]*SIGNAL_SENSOR_5[1]+FC_MATRIX_Y[6]*SIGNAL_SENSOR_6[1]+FC_MATRIX_Y[7]*SIGNAL_SENSOR_7[1]+FC_MATRIX_Y[8]*SIGNAL_SENSOR_8[1]+FC_MATRIX_Y[9]*SIGNAL_SENSOR_9[1]+FC_MATRIX_Y[10]*SIGNAL_SENSOR_10[1]);
FORCE_ROW[3]:=(FC_MATRIX_Z[1]*SIGNAL_SENSOR_1[1]+FC_MATRIX_Z[2]*SIGNAL_SENSOR_2[1]+FC_MATRIX_Z[3]*SIGNAL_SENSOR_3[1]+FC_MATRIX_Z[4]*SIGNAL_SENSOR_4[1]+FC_MATRIX_Z[5]*SIGNAL_SENSOR_5[1]+FC_MATRIX_Z[6]*SIGNAL_SENSOR_6[1]+FC_MATRIX_Z[7]*SIGNAL_SENSOR_7[1]+FC_MATRIX_Z[8]*SIGNAL_SENSOR_8[1]+FC_MATRIX_Z[9]*SIGNAL_SENSOR_9[1]+FC_MATRIX_Z[10]*SIGNAL_SENSOR_10[1]);

IF FORCE_RESET>0 THEN
	FORCE_SUM[1]:=FORCE_ROW[1]+FORCE_SUM[1];
	FORCE_SUM[2]:=FORCE_ROW[2]+FORCE_SUM[2];
	FORCE_SUM[3]:=FORCE_ROW[3]+FORCE_SUM[3];
	INK:=INK+1;
	IF INK=1000 THEN
		RESET_FORCE_VAL[1]:=FORCE_SUM[1]/INK;
		RESET_FORCE_VAL[2]:=FORCE_SUM[2]/INK;
		RESET_FORCE_VAL[3]:=FORCE_SUM[3]/INK;
		INK:=0;
		FORCE_RESET:=0;
		FORCE_SUM[1]:=0;
		FORCE_SUM[2]:=0;
		FORCE_SUM[3]:=0;
	END_IF
END_IF


SIGNAL_FORCE[1]:=FORCE_ROW[1]-RESET_FORCE_VAL[1];
SIGNAL_FORCE[2]:=FORCE_ROW[2]-RESET_FORCE_VAL[2];
SIGNAL_FORCE[3]:=FORCE_ROW[3]-RESET_FORCE_VAL[3];

FILTER_FX(ssMethodType:=1 , IN:= SIGNAL_FORCE[1], OUT=> SIGNAL_FORCE_FLT[1]);
FILTER_FY(ssMethodType:=1 , IN:= SIGNAL_FORCE[2], OUT=> SIGNAL_FORCE_FLT[2]);
FILTER_FZ(ssMethodType:=1 , IN:= SIGNAL_FORCE[3], OUT=> SIGNAL_FORCE_FLT[3]);

END_PROGRAM

// ---- POUs/DEFLECTION_CONTROL_FEED.TcPOU
PROGRAM DEFLECTION_CONTROL_FEED
VAR
		USED_FORCE_SIGNAL: REAL:=0;
		DEFLECTION_REAL: REAL:=0;
END_VAR

IF ACT_NC_PROGRAM=5 THEN
	
	//USED_FORCE_SIGNAL:=-A_SIGNAL_2;
	//USED_FORCE_SIGNAL:=SIGNAL_FORCE_FLT[2];
	USED_FORCE_SIGNAL:=SQRT(EXPT(A_SIGNAL_1,2)+EXPT(A_SIGNAL_2,2));
		
	IF USED_FORCE_SIGNAL<0 THEN
		FORCE_ACT:=0;
		ELSE FORCE_ACT:=USED_FORCE_SIGNAL;	
	END_IF
	
	
	TOOL_STIFFNESS_ACT:=TOOL_STIFFNESS_SELC_PTS[1,3];
	//TOOL_STIFFNESS_ACT:=TOOL_STIFFNESS_SELC_PTS[2,3];
	DEFLECTION_ACT:=FORCE_ACT/TOOL_STIFFNESS_ACT;		//µm
		
	
	IF ACT_NC_PROGRAM_STEP=1 THEN
			DEFLECTION_CONTROL_ON:=1;			//DEFLECTION CONTROL ON		
		ELSE
			DEFLECTION_CONTROL_ON:=0;
	END_IF

	IF DEFLECTION_CONTROL_ON=0 THEN
		CONTROL_RESET:=1;
	END_IF

	IF DEFLECTION_CONTROL_ON=1 AND CONTROL_RESET=1 THEN
		DEFLECTION_DIF_SUM:=0;
		CUTTING_ON:=0;
		REF_REACHED:=0;
		CONTROL_RESET:=0;
	END_IF

	CASE ACT_NC_PARAM_3 OF					// CONTROL STRUCTURE SELECT 
		1:
			CONTROLLER_TYPE:=1;				// P CONTROLLER
		2:
			CONTROLLER_TYPE:=2;				// PI CONTROLLER 
		3:
			CONTROLLER_TYPE:=3;				// PI CONTROLLER WITH ANTI-WINDUP
		ELSE
			CONTROLLER_TYPE:=1;				// P CONTROLLER
	END_CASE

	IF FORCE_ACT>=CUTTING_FORCE_MIN AND CUTTING_ON=0 THEN
		CUTTING_ON:=1;
	END_IF
	
	IF DEFLECTION_ACT>=DEFLECTION_REF AND REF_REACHED=0 THEN
		REF_REACHED:=1;
	END_IF

	CASE ACT_NC_PARAM_4 OF					// START CONDITION SELECTION FOR CONTROLLER
		1:
			CONTROL_START:=1;
			CONTROL_START_CONDITION:=(DEFLECTION_CONTROL_ON=1);				        //CONDITION CONTROL ON
		2:
			CONTROL_START:=2;
			CONTROL_START_CONDITION:=(DEFLECTION_CONTROL_ON=1 AND CUTTING_ON=1);	//CONDITION CUTTING ON
		3:
			CONTROL_START:=3;
			CONTROL_START_CONDITION:=(DEFLECTION_CONTROL_ON=1 AND REF_REACHED=1);	//CONDITION REF REACHED
		ELSE
			CONTROL_START:=1;
			CONTROL_START_CONDITION:=(DEFLECTION_CONTROL_ON=1);
	END_CASE

	IF CONTROL_START_CONDITION=1 THEN
	
		DEFLECTION_DIF:=DEFLECTION_REF-DEFLECTION_ACT;
	
		IF CONTROLLER_TYPE=1 THEN
			OVRD_REG_P:=K_P*DEFLECTION_DIF;
			OVRD_REG_I:=0;
		END_IF
	
		IF CONTROLLER_TYPE=2 THEN
			DEFLECTION_DIF_SUM:=DEFLECTION_DIF_SUM+DEFLECTION_DIF;
			OVRD_REG_P:=K_P*DEFLECTION_DIF;
			OVRD_REG_I:=K_I*T_S*DEFLECTION_DIF_SUM;
		END_IF
	
		IF CONTROLLER_TYPE=3 THEN
			OVRD_DIF:=OVRD_REG-OVRD_MACHINE;
			WINDUP:=K_WINDUP*OVRD_DIF;
			DEFLECTION_DIF_SUM:=DEFLECTION_DIF_SUM+K_I*T_S*DEFLECTION_DIF-WINDUP;
			OVRD_REG_P:=K_P*DEFLECTION_DIF;
			OVRD_REG_I:=DEFLECTION_DIF_SUM;	
		END_IF
		
		OVRD_REG:=OVRD_REG_P+OVRD_REG_I+OVRD_MID;
		OVRD_MACHINE:=OVRD_REG;
	
		IF OVRD_MACHINE > SATURATION_OVRD_MAX THEN
			OVRD_MACHINE:=SATURATION_OVRD_MAX;
		END_IF

		IF OVRD_MACHINE < SATURATION_OVRD_MIN THEN
			OVRD_MACHINE:=SATURATION_OVRD_MIN;
		END_IF
	
		ELSE OVRD_MACHINE:=OVRD_MID;
	
	END_IF
		
	SET_NC_PARAM_2:= REAL_TO_WORD(OVRD_MACHINE);
	ELSE
		SET_NC_PARAM_2:= 100;
END_IF

END_PROGRAM

// ---- POUs/TOUCH_PROBE_LINE.TcPOU
PROGRAM TOUCH_PROBE_LINE
VAR
	IND_MEAS:		WORD:=0;
	i:				WORD:=1;
	reset:			WORD:=0;
END_VAR

IF ACT_NC_PROGRAM=20 THEN	//NC-PROGRAM NUMBER FOR TOUCH_PROBE_LINE
	
	IND_MEAS:=ACT_NC_PROGRAM_STEP;
		
	IF IND_MEAS=1000 THEN
		FOR i:=1 TO 50 DO
			PTS_POSITION[i]:=0;
			PTS_MEASUREMENT[i]:=0;
		END_FOR
		FOR i:=1 TO 10 DO
			PTS_MEASUREMENT_HISTOGRAM_1[i]:=0;
			PTS_MEASUREMENT_HISTOGRAM_2[i]:=0;
		END_FOR
		RESULT[0]:=0;
		RESULT[1]:=0;
	END_IF
	
	IF IND_MEAS=1001 THEN
		FOR i:=1 TO 50 DO
			PTS_POSITION[i]:=0;
			PTS_MEASUREMENT[i]:=0;
		END_FOR
		FOR i:=1 TO 10 DO
			PTS_MEASUREMENT_HISTOGRAM_2[i]:=0;
		END_FOR
		RESULT[1]:=0;
	
	END_IF
	
	IF IND_MEAS<>0 AND IND_MEAS<=100 AND(IND_MEAS MOD 2)=1 THEN 
		PTS_POSITION[(IND_MEAS+1)/2]:=ACT_NC_PARAM_5;	
	END_IF
	
	IF IND_MEAS<>0 AND IND_MEAS<=100 AND(IND_MEAS MOD 2)=0 THEN 
		PTS_MEASUREMENT[IND_MEAS/2]:=ACT_NC_PARAM_5;
	END_IF
	
	IF IND_MEAS=2000 THEN
		FOR i:=1 TO 10 DO
			//PTS_MEASUREMENT_HISTOGRAM_1[i]:=0;
			//PTS_MEASUREMENT_HISTOGRAM_1[i]:=PTS_MEASUREMENT[PTS_SELCT_HISTOGRAM[i]];
			PTS_MEASUREMENT_HISTOGRAM_1[i]:=1000*(PTS_MEASUREMENT[PTS_SELCT_HISTOGRAM[i]]-PTS_MEASUREMENT[1]);
		END_FOR
		RESULT[0]:=ABS(PTS_MEASUREMENT_HISTOGRAM_1[2]);
	END_IF
	
	IF IND_MEAS=3000 THEN
		FOR i:=1 TO 10 DO
			//PTS_MEASUREMENT_HISTOGRAM_2[i]:=0;
			//PTS_MEASUREMENT_HISTOGRAM_2[i]:=PTS_MEASUREMENT[PTS_SELCT_HISTOGRAM[i]];
			PTS_MEASUREMENT_HISTOGRAM_2[i]:=1000*(PTS_MEASUREMENT[PTS_SELCT_HISTOGRAM[i]]-PTS_MEASUREMENT[1]);
		END_FOR
		IF ABS(PTS_MEASUREMENT_HISTOGRAM_2[2])>6 THEN
			RESULT[1]:=ABS(PTS_MEASUREMENT_HISTOGRAM_2[2])/2.5;
			ELSE
				RESULT[1]:=ABS(PTS_MEASUREMENT_HISTOGRAM_2[2]);
		END_IF
		//RESULT[1]:=ABS(PTS_MEASUREMENT_HISTOGRAM_2[2]);
	END_IF
	
END_IF

END_PROGRAM

// ---- POUs/DP_CONFIG_OUT_EL6731.TcPOU
PROGRAM DP_CONFIG_OUT_EL6731
VAR
END_VAR

DP_MISO_WORD_1:=SET_NC_PARAM_1;	
DP_MISO_WORD_2:=SET_NC_PARAM_2;
DP_MISO_WORD_3:=SET_NC_PARAM_3;													
DP_MISO_WORD_4:=SET_NC_PARAM_4;

END_PROGRAM

// ---- POUs/ADAS_Kom.TcPOU
PROGRAM ADAS_Kom
VAR CONSTANT
	///defaultConfig : AdasConfiguration := (track := [1, 2, 3, 4, 5, 6, 7, 8, 9, 10, 11, 12, 13, 14, 15, 16, 17, 18, 19, 20, 21, 22, 23, 24, 25, 26, 27, 28, 29, 30],
	///										signal:= [4, 4, 4, 4, 4, 5, 5, 5, 5,  5,  5,  6,  6,  6,  6,  6,  6, 17, 17, 17, 17, 17, 17,  1,  1,  1,  1,  1,  1,  1],
	///										axis  := [1, 1, 2, 3, 4, 1, 1, 2, 3,  4,  5,  1,  1,  2,  3,  4,  5,  1,  1,  2,  3,  4,  5,  1,  1,  2,  3,  4,  5,  1]);
	///
	///
	///unten stehende Konfiguration nach neuen Schema
	///1->6
	///2->1
	///3->2
	///4->3
	///5->4
	///6->1
	///
	///											Messwert	Position		Geschwindigkeit				Beschleunigung				Strom						Offen
	///											Funktion x, x, x, x, o, 	x, x, x, x,  x,  ?,		 x,  x,  x,  x,  x,  ?,		 x,  x,  x,  x,  x,  ?,	
	///											Achse	 x, y, z, c, n, 	x, y, z, c,  b,  n, 	 x,  y,  z,  c,  b,  n,		 x,  y,  z,  c,  b,  n,
	defaultConfig: AdasConfiguration := (track := [1, 2, 3, 4, 5, 6, 7, 8, 9, 10, 11, 12, 13, 14, 15, 16, 17, 18, 19, 20, 21, 22, 23, 24, 25, 26, 27, 28, 29, 30], signal := [4, 4, 4, 4, 4, 5, 5, 5, 5, 5, 5, 6, 6, 6, 6, 6, 6, 17, 17, 17, 17, 17, 17, 4, 4, 1, 1, 1, 1, 1], axis := [6, 1, 2, 3, 4, 6, 1, 2, 3, 4, 5, 6, 1, 2, 3, 4, 5, 6, 1, 2, 3, 4, 5, 6, 5, 6, 6, 1, 1, 1]);
	/// Lesen von allen 30 Datenstreams
	numberOfDefaultTracks: UINT := 30;
	/// Anzahl ms die nach Ausgabe einer Anforderung gewartet werden soll, bevor die Antwort ausgewertet wird.
	waitTime: INT := 50;
END_VAR
VAR_INPUT
	ADAS_IN AT %I*: ARRAY[0..63] OF WORD;
	/// UNION  aus DUTs
	adasStream_IN: AdasData_In;
	/// STRUCT aus DUTs
	requestedConfiguration_IN AT %I*: AdasConfiguration;
	numberOfRequestetTracks_IN AT %I*: UINT;
	ConfigRequest_IN AT %I*: BOOL;
END_VAR
VAR
	waitTimer: INT := 0;
	/// STRUCT aus DUTs
	actualConfig: AdasConfiguration;
	/// STRUCT aus DUTs
	requestedConfiguration: AdasConfiguration;
	configRequestTrigger: R_TRIG;
	tracksToConfig: UINT;
	configuredTracks: UINT := 0;
	index: UINT;
	///ENUM aus DUTs
	comState: eAdasKom_State := eAdasKom_State.WaitForNC;
	///ENUM aus DUTs
	configState: eAdasKonfig_State := eAdasKonfig_State.Init;
	selectCounter: SINT := 0;
	init: BOOL := 0;
	kommzeit: BOOL := 0;
	deint: BOOL := 0;
	track: BOOL := 0;
	signal: BOOL := 0;
END_VAR
VAR_OUTPUT
	/// UNION  aus DUTs
	adasStreamSetup_OUT AT %Q*: AdasSetup_Out;
	adasData AT %Q*: ARRAY[0..(gVarL.gVar_NumberOfAdasTracks - 1)] OF DINT;
	StartExe: INT;
END_VAR

adasStream_IN.asBin := ADAS_IN;

//Kommunikationszykluszeit von ADAS festlegen
IF kommzeit THEN
	//The machine axes numbers basically range from 1 to 31. Only axes that are enabled by 20070 $MC_AXCONF_MACHAX_USED within one of the active channels can supply data.
	adasStreamSetup_OUT.asSetup.blockType   := 15;	//entspricht 0xF aus Anleitung
	adasStreamSetup_OUT.asSetup.blockLength := 8;	//festgelegt in Anleitung
	adasStreamSetup_OUT.asSetup.selectTrack := 255; //Command mode
	adasStreamSetup_OUT.asSetup.selectAxis  := 100; //wenn man zykluszeit wechseln will
	adasStreamSetup_OUT.asSetup.selectSignal:= 8; //neue zykluszeit: 10x 0.5ms =5ms
	adasStreamSetup_OUT.asSetup.selectFlag  := adasStream_IN.asData.acceptFlag;
	kommzeit := 0;
	comState := eAdasKom_State.WaitForNC;
	configState := eAdasKonfig_State.Init;
END_IF


//Track bezeichnung senden von ADAS-Kommunikation
IF track THEN
	//The machine axes numbers basically range from 1 to 31. Only axes that are enabled by 20070 $MC_AXCONF_MACHAX_USED within one of the active channels can supply data.
	adasStreamSetup_OUT.asSetup.blockType   := 15;	//entspricht 0xF aus Anleitung
	adasStreamSetup_OUT.asSetup.blockLength := 8;	//festgelegt in Anleitung
	adasStreamSetup_OUT.asSetup.selectTrack := 255; //Comande mode
	adasStreamSetup_OUT.asSetup.selectAxis  := 122; //all tracks resetten
	adasStreamSetup_OUT.asSetup.selectSignal:= 0;   //Vorgabe
	adasStreamSetup_OUT.asSetup.selectFlag  := adasStream_IN.asData.acceptFlag;
	track := 0;
	comState := eAdasKom_State.WaitForNC;
	configState := eAdasKonfig_State.Init;
END_IF

//Signal bezeichnung senden von ADAS-Kommunikation
IF signal THEN
	//The machine axes numbers basically range from 1 to 31. Only axes that are enabled by 20070 $MC_AXCONF_MACHAX_USED within one of the active channels can supply data.
	adasStreamSetup_OUT.asSetup.blockType   := 15;	//entspricht 0xF aus Anleitung
	adasStreamSetup_OUT.asSetup.blockLength := 8;	//festgelegt in Anleitung
	adasStreamSetup_OUT.asSetup.selectTrack := 255; //Comande mode
	adasStreamSetup_OUT.asSetup.selectAxis  := 123; //all tracks resetten
	adasStreamSetup_OUT.asSetup.selectSignal:= 0;   //Vorgabe
	adasStreamSetup_OUT.asSetup.selectFlag  := adasStream_IN.asData.acceptFlag;
	signal := 0;
	comState := eAdasKom_State.WaitForNC;
//	configState := eAdasKonfig_State.Init;
END_IF


//Deinitialisierung von ADAS-Kommunikation
IF deint THEN
	//The machine axes numbers basically range from 1 to 31. Only axes that are enabled by 20070 $MC_AXCONF_MACHAX_USED within one of the active channels can supply data.
	adasStreamSetup_OUT.asSetup.blockType   := 15;	//entspricht 0xF aus Anleitung
	adasStreamSetup_OUT.asSetup.blockLength := 8;	//festgelegt in Anleitung
	adasStreamSetup_OUT.asSetup.selectTrack := 255; //Comande mode
	adasStreamSetup_OUT.asSetup.selectAxis  := 110; //all tracks resetten
	adasStreamSetup_OUT.asSetup.selectSignal:= 0;   //Vorgabe
	adasStreamSetup_OUT.asSetup.selectFlag  := adasStream_IN.asData.acceptFlag;
	deint := 0;
	comState := eAdasKom_State.WaitForNC;
	configState := eAdasKonfig_State.Init;
END_IF

//Initialisierung von ADAS-Kommunikation
IF init THEN
	//The machine axes numbers basically range from 1 to 31. Only axes that are enabled by 20070 $MC_AXCONF_MACHAX_USED within one of the active channels can supply data.
	adasStreamSetup_OUT.asSetup.blockType   := 15;	//entspricht 0xF aus Anleitung
	adasStreamSetup_OUT.asSetup.blockLength := 8;	//festgelegt in Anleitung
	adasStreamSetup_OUT.asSetup.selectTrack := 0;
	adasStreamSetup_OUT.asSetup.selectAxis  := 0;
	adasStreamSetup_OUT.asSetup.selectSignal:= 0;
	adasStreamSetup_OUT.asSetup.selectFlag  := adasStream_IN.asData.acceptFlag;
	init := 0;
	comState := eAdasKom_State.WaitForNC;
	configState := eAdasKonfig_State.Init;
END_IF




CASE comState OF
	eAdasKom_State.WaitForNC:
		IF adasStream_IN.asData.comCycle > 0 THEN
			comState := eAdasKom_State.SetDefaultkonfig;
			requestedConfiguration := defaultConfig;
			tracksToConfig := numberOfDefaultTracks;
			configState := eAdasKonfig_State.SendTrackConfig;
			configuredTracks := 0;		
		END_IF
		
	eAdasKom_State.SetDefaultkonfig:
		CASE configState OF
			eAdasKonfig_State.SendTrackConfig:
			    selectCounter := adasStream_IN.asData.acceptFlag;
				selectCounter := selectCounter + 1;
				IF (selectCounter > 127) THEN
					selectCounter := 0;
				END_IF
				adasStreamSetup_OUT.asSetup.selectAxis 	:= requestedConfiguration.axis[configuredTracks];
				adasStreamSetup_OUT.asSetup.selectSignal:= requestedConfiguration.signal[configuredTracks];
				adasStreamSetup_OUT.asSetup.selectTrack	:= requestedConfiguration.track[configuredTracks];
				adasStreamSetup_OUT.asSetup.selectFlag	:= selectCounter;
				configState := eAdasKonfig_State.WaitForSelectFlag;
				waitTimer := 0;
			eAdasKonfig_State.WaitForSelectFlag:
				waitTimer := waitTimer + 1;
				IF (waitTimer >= waitTime)THEN
					IF (adasStream_IN.asData.acceptFlag = selectCounter)THEN
						
						actualConfig.axis[requestedConfiguration.track[configuredTracks] - 1]  := requestedConfiguration.axis[configuredTracks];
						actualConfig.signal[requestedConfiguration.track[configuredTracks]- 1] := requestedConfiguration.signal[configuredTracks];
						actualConfig.track[requestedConfiguration.track[configuredTracks] - 1] := requestedConfiguration.track[configuredTracks];
						
						configuredTracks := configuredTracks + 1;
						IF configuredTracks = tracksToConfig THEN
							comState :=	eAdasKom_State.Running;
							configState := eAdasKonfig_State.ConfigCurrent;
						ELSE
							configState := eAdasKonfig_State.SendTrackConfig;
						END_IF
	
					ELSIF (adasStream_IN.asData.acceptFlag < 0) THEN
						comState :=	eAdasKom_State.Error;		
					END_IF
				END_IF
		END_CASE
				
	eAdasKom_State.Running:
		adasData := adasStream_IN.asData.Data;
		CASE configState OF 
			eAdasKonfig_State.ConfigCurrent:
				configRequestTrigger(CLK := ConfigRequest_IN);
				IF configRequestTrigger.Q THEN
					requestedConfiguration := requestedConfiguration_IN;
					tracksToConfig := numberOfRequestetTracks_IN;
					configuredTracks := 0;
					configState := eAdasKonfig_State.SendTrackConfig;
				END_IF
			eAdasKonfig_State.SendTrackConfig:
				selectCounter := adasStream_IN.asData.acceptFlag;
				selectCounter := selectCounter + 1;
				IF (selectCounter > 127) THEN
					selectCounter := 0;
				END_IF
				adasStreamSetup_OUT.asSetup.selectAxis 	:= requestedConfiguration.axis[configuredTracks];
				adasStreamSetup_OUT.asSetup.selectSignal:= requestedConfiguration.signal[configuredTracks];
				adasStreamSetup_OUT.asSetup.selectTrack	:= requestedConfiguration.track[configuredTracks];
				adasStreamSetup_OUT.asSetup.selectFlag	:= selectCounter;
				configState := eAdasKonfig_State.WaitForSelectFlag;
			eAdasKonfig_State.WaitForSelectFlag:
				IF (adasStream_IN.asData.acceptFlag = selectCounter)THEN
					
					actualConfig.axis[requestedConfiguration.track[configuredTracks]]   := requestedConfiguration.axis[configuredTracks];
					actualConfig.signal[requestedConfiguration.track[configuredTracks]] := requestedConfiguration.signal[configuredTracks];
					actualConfig.track[requestedConfiguration.track[configuredTracks]]  := requestedConfiguration.track[configuredTracks];
					
					configuredTracks := configuredTracks + 1;
					IF configuredTracks = tracksToConfig THEN
						configState := eAdasKonfig_State.ConfigCurrent;
					ELSE
						configState := eAdasKonfig_State.SendTrackConfig;
					END_IF
				ELSIF (adasStream_IN.asData.acceptFlag < 0) THEN
					comState :=	eAdasKom_State.Error;		
				END_IF
		END_CASE
	eAdasKom_State.Error:	
END_CASE

END_PROGRAM

// ---- VISUs/VISUALISATION_DEFLEC_CONTROL.TcVIS
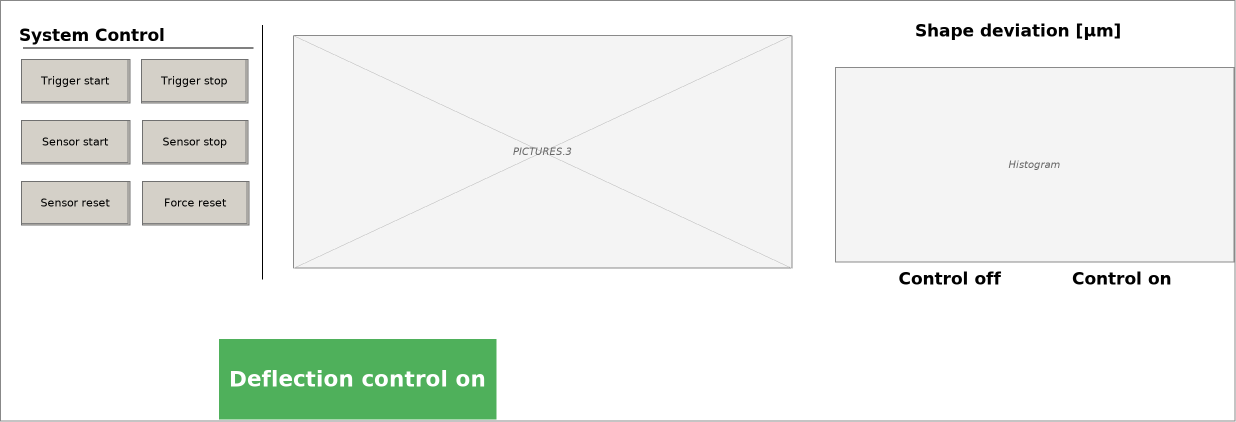
VISUALIZATION VISUALISATION_DEFLEC_CONTROL  // 1236x422
    Button (21,59 109x44), "Trigger start"
        OnMouseClick: execute { VARIABLES.CAN_TRIGGER_STATE:=1; }
    Button (141,59 107x44), "Trigger stop"
        OnMouseClick: execute { VARIABLES.CAN_TRIGGER_STATE:=0; }
    Button (21,120 109x44), "Sensor start"
        OnMouseClick: execute { CAN_CONTROL_STATE:=1; }
    Button (142,120 106x44), "Sensor stop"
        OnMouseClick: execute { CAN_CONTROL_STATE:=0; }
    Button (21,181 109x44), "Sensor reset"
        OnMouseClick: execute { CAN_CONTROL_STATE:=2; }
    Button (142,181 107x44), "Force reset"
        OnMouseClick: execute { VARIABLES.FORCE_RESET:=1; }
    Rectangle (17,20 150x30), "System Control"
    Line (253,48) (23,48)
    Rectangle (1056,265 132x27), "Control on"
    Rectangle (871,265 158x27), "Control off"
    Line (262,25) (262,279)
    Rectangle (896,17 245x27), "Shape deviation [µm]"
    Image (293,35 499x233), image: PICTURES.3
    Histogram (835,67 399x195), scale format: %.1f, scale 0..60
        p1518820177: VARIABLES.RESULT
        p102497268: VARIABLES.RESULT
        p788070771: ARRAY [0..1] OF REAL
    Rectangle (218,338 279x82), "Deflection control on", invisible if: DEFLECTION_CONTROL_ON<>1
END_VISUALIZATION

// ---- VISUs/VISUALISATION_EMO2017.TcVIS
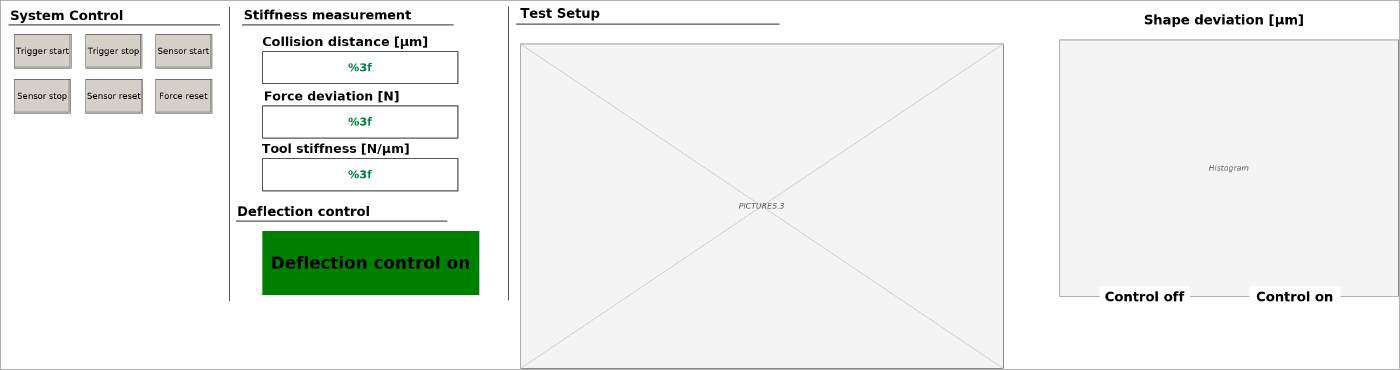
VISUALIZATION VISUALISATION_EMO2017  // 1804x477
    Rectangle (338,298 279x82), "Deflection control off", invisible if: 1
    Button (18,44 74x44), "Trigger start"
        OnMouseClick: execute { VARIABLES.CAN_TRIGGER_STATE:=1; }
    Button (110,44 73x44), "Trigger stop"
        OnMouseClick: execute { VARIABLES.CAN_TRIGGER_STATE:=0; }
    Button (200,44 73x44), "Sensor start"
        OnMouseClick: execute { CAN_CONTROL_STATE:=1; }
    Button (18,102 73x44), "Sensor stop"
        OnMouseClick: execute { CAN_CONTROL_STATE:=0; }
    Button (110,102 74x44), "Sensor reset"
        OnMouseClick: execute { CAN_CONTROL_STATE:=2; }
    Button (200,102 73x44), "Force reset"
        OnMouseClick: execute { FORCE_RESET:=1; }
    Rectangle (11,5 150x30), "System Control"
    Rectangle (313,12 218x15), "Stiffness measurement"
    Rectangle (338,204 252x42), "%3f", text variable: VARIABLES.TOOL_STIFFNESS[1]
    Rectangle (338,66 252x42), "%3f", text variable: VARIABLES.COLLISION_DISTANCE
    Rectangle (338,136 252x42), "%3f", text variable: VARIABLES.FORCE_DEVIATION[1]
    Rectangle (337,44 216x20), "Collision distance [µm]"
    Rectangle (340,114 175x20), "Force deviation [N]"
    Rectangle (338,183 190x17), "Tool stiffness [N/µm]"
    Line (295,9) (295,388)
    Line (584,32) (312,32)
    Group (1365,12 437x384)
        Histogram (0,39 437x331), scale format: %.1f, scale 0..50
            p1518820177: VARIABLES.RESULT
            p102497268: VARIABLES.RESULT
            p788070771: ARRAY [1..2] OF REAL
        Rectangle (245,357 117x27), "Control on"
        Rectangle (52,357 116x27), "Control off"
        Rectangle (110,0 205x27), "Shape deviation [µm]"
    Line (283,32) (11,32)
    Image (670,56 623x419), image: PICTURES.3
    Rectangle (654,-2 136x38), "Test Setup"
    Line (1004,31) (665,31)
    Line (655,8) (655,387)
    Line (576,285) (304,285)
    Rectangle (301,265 181x15), "Deflection control"
    Rectangle (338,298 279x82), "Deflection control on", invisible if: DEFLECTION_CONTROL_ON<>1
END_VISUALIZATION

// ---- VISUs/VISUALISATION_SENSOR_CONTROL.TcVIS
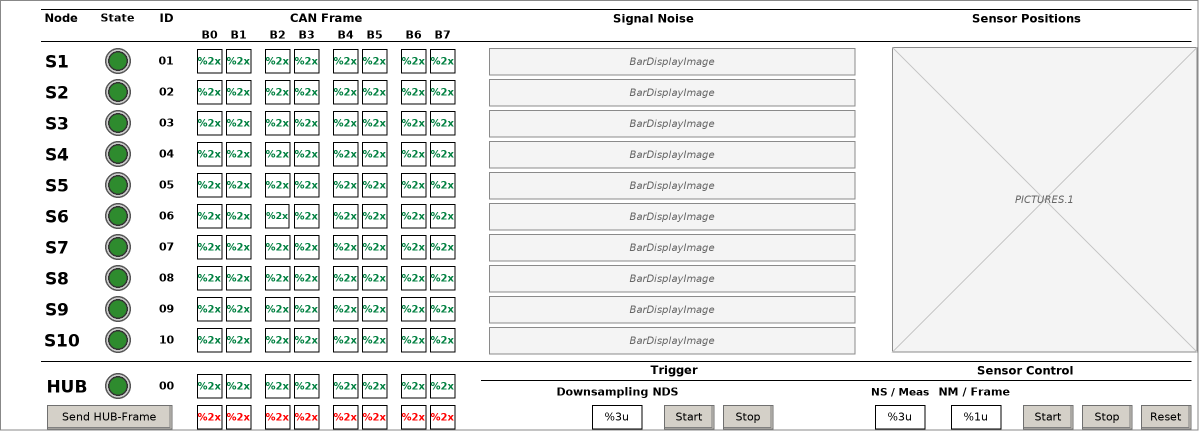
VISUALIZATION VISUALISATION_SENSOR_CONTROL  // 1199x431
    Group (870,363 321x66)
        Rectangle (65,17 79x24), "NM / Frame"
        Rectangle (0,17 61x24), "NS / Meas"
        Button (153,42 50x24), "Start"
            OnMouseClick: execute { CAN_CONTROL_STATE:=1; }
        Button (212,42 50x24), "Stop"
            OnMouseClick: execute { CAN_CONTROL_STATE:=0; }
        Button (271,42 50x24), "Reset"
            OnMouseClick: execute { CAN_CONTROL_STATE:=2; }
        Rectangle (81,42 50x24), "%1u", text variable: VARIABLES.M_PER_FRAME
            OnMouseDown: write the text variable via Default, min 0, max 4
        Rectangle (97,0 117x15), "Sensor Control"
        Rectangle (5,42 50x24), "%3u", text variable: VARIABLES.N_SAMPLES_PER_M
            OnMouseDown: write the text variable via Default, min 0, max 255
    Group (507,359 266x70)
        Rectangle (97,0 140x22), "Trigger"
        Button (157,46 50x24), "Start"
            OnMouseClick: execute { VARIABLES.CAN_TRIGGER_STATE:=1; }
        Rectangle (0,21 221x24), "Downsampling NDS"
        Rectangle (85,46 50x24), "%3u", text variable: VARIABLES.K_TRIGGER
            OnMouseDown: write the text variable via Default
        Button (216,46 50x24), "Stop"
            OnMouseClick: execute { VARIABLES.CAN_TRIGGER_STATE:=0; }
    Group (489,11 366x343)
        BarDisplayImage (0,37 366x27), value: VARIABLES.SIGNAL_DEVIATION[1], style: BarDisplayImage-Gray, scale format: %1u, scale 0..200
        BarDisplayImage (0,68 366x27), value: VARIABLES.SIGNAL_DEVIATION[2], style: BarDisplayImage-Gray, scale format: %1u, scale 0..200
        BarDisplayImage (0,99 366x27), value: VARIABLES.SIGNAL_DEVIATION[3], style: BarDisplayImage-Gray, scale format: %1u, scale 0..200
        BarDisplayImage (0,130 366x27), value: VARIABLES.SIGNAL_DEVIATION[4], style: BarDisplayImage-Gray, scale format: %1u, scale 0..200
        BarDisplayImage (0,161 366x27), value: VARIABLES.SIGNAL_DEVIATION[5], style: BarDisplayImage-Gray, scale format: %1u, scale 0..200
        BarDisplayImage (0,192 366x27), value: VARIABLES.SIGNAL_DEVIATION[6], style: BarDisplayImage-Gray, scale format: %1u, scale 0..200
        BarDisplayImage (0,223 366x27), value: VARIABLES.SIGNAL_DEVIATION[7], style: BarDisplayImage-Gray, scale format: %1u, scale 0..200
        Rectangle (106,0 117x15), "Signal Noise"
        BarDisplayImage (0,254 366x27), value: VARIABLES.SIGNAL_DEVIATION[8], style: BarDisplayImage-Gray, scale format: %1u, scale 0..200
        BarDisplayImage (0,285 366x27), value: VARIABLES.SIGNAL_DEVIATION[9], style: BarDisplayImage-Gray, scale format: %1u, scale 0..200
        BarDisplayImage (0,316 366x27), value: VARIABLES.SIGNAL_DEVIATION[10], style: BarDisplayImage-Gray, scale format: %1u, scale 0..200
    Group (29,371 426x58)
        Button (18,34 125x24), "Send HUB-Frame"
            OnMouseClick: execute { CAN_CONTROL_STATE:=3; }
        Rectangle (401,34 25x24), "%2x", text variable: VARIABLES.CAN_PARAMETER_FRAME[7]
            OnMouseDown: write the text variable via Default
        Rectangle (372,34 25x24), "%2x", text variable: VARIABLES.CAN_PARAMETER_FRAME[6]
            OnMouseDown: write the text variable via Default
        Rectangle (333,34 25x24), "%2x", text variable: VARIABLES.CAN_PARAMETER_FRAME[5]
            OnMouseDown: write the text variable via Default
        Rectangle (304,34 25x24), "%2x", text variable: VARIABLES.CAN_PARAMETER_FRAME[4]
            OnMouseDown: write the text variable via Default
        Rectangle (265,34 25x24), "%2x", text variable: VARIABLES.CAN_PARAMETER_FRAME[3]
            OnMouseDown: write the text variable via Default
        Rectangle (236,34 25x24), "%2x", text variable: VARIABLES.CAN_PARAMETER_FRAME[2]
            OnMouseDown: write the text variable via Default
        Rectangle (197,34 25x24), "%2x", text variable: VARIABLES.CAN_PARAMETER_FRAME[1]
            OnMouseDown: write the text variable via Default
        Rectangle (168,34 25x24), "%2x", text variable: VARIABLES.CAN_PARAMETER_FRAME[0]
            OnMouseDown: write the text variable via Default
        Rectangle (0,2 76x27), "HUB"
        Lamp1 (74,0 30x30), variable: VARIABLES.HUB_STATE, style: Lamp-Lamp1-Green
        Rectangle (168,3 25x24), "%2x", text variable: VARIABLES.CAN_HUB [0]
        Rectangle (197,3 25x24), "%2x", text variable: VARIABLES.CAN_HUB [1]
        Rectangle (236,3 25x24), "%2x", text variable: VARIABLES.CAN_HUB [2]
        Rectangle (265,3 25x24), "%2x", text variable: VARIABLES.CAN_HUB [3]
        Rectangle (304,3 25x24), "%2x", text variable: VARIABLES.CAN_HUB [4]
        Rectangle (333,3 25x24), "%2x", text variable: VARIABLES.CAN_HUB [5]
        Rectangle (372,3 25x24), "%2x", text variable: VARIABLES.CAN_HUB [6]
        Rectangle (401,3 25x24), "%2x", text variable: VARIABLES.CAN_HUB [7]
        Rectangle (125,3 25x24), "00"
    Group (19,13 436x342)
        Rectangle (0,35 76x27), "S1"
        Rectangle (0,66 76x27), "S2"
        Rectangle (0,97 76x27), "S3"
        Rectangle (0,128 76x27), "S4"
        Rectangle (0,159 76x27), "S5"
        Rectangle (0,190 76x27), "S6"
        Rectangle (0,221 76x27), "S7"
        Rectangle (0,252 76x27), "S8"
        Rectangle (0,283 76x27), "S9"
        Lamp1 (84,33 30x30), variable: VARIABLES.SENSOR_STATE[1], style: Lamp-Lamp1-Green
        Lamp1 (84,64 30x30), variable: VARIABLES.SENSOR_STATE[2], style: Lamp-Lamp1-Green
        Lamp1 (84,95 30x30), variable: VARIABLES.SENSOR_STATE[3], style: Lamp-Lamp1-Green
        Lamp1 (84,126 30x30), variable: VARIABLES.SENSOR_STATE[4], style: Lamp-Lamp1-Green
        Lamp1 (84,157 30x30), variable: VARIABLES.SENSOR_STATE[5], style: Lamp-Lamp1-Green
        Lamp1 (84,188 30x30), variable: VARIABLES.SENSOR_STATE[6], style: Lamp-Lamp1-Green
        Lamp1 (84,219 30x30), variable: VARIABLES.SENSOR_STATE[7], style: Lamp-Lamp1-Green
        Rectangle (178,10 25x24), "B0"
        Rectangle (207,10 25x24), "B1"
        Rectangle (246,10 25x24), "B2"
        Rectangle (275,10 25x24), "B3"
        Rectangle (314,10 25x24), "B4"
        Rectangle (343,10 25x24), "B5"
        Rectangle (382,10 25x24), "B6"
        Rectangle (411,10 25x24), "B7"
        Rectangle (270,0 75x10), "CAN Frame"
        Rectangle (130,0 35x10), "ID"
        Rectangle (18,0 49x10), "Node"
        Rectangle (81,0 35x10), "State"
        Lamp1 (84,250 30x30), variable: VARIABLES.SENSOR_STATE[8], style: Lamp-Lamp1-Green
        Lamp1 (84,281 30x30), variable: VARIABLES.SENSOR_STATE[9], style: Lamp-Lamp1-Green
        Rectangle (5,314 76x27), "S10"
        Lamp1 (84,312 30x30), variable: VARIABLES.SENSOR_STATE[10], style: Lamp-Lamp1-Green
        Rectangle (178,36 25x24), "%2x", text variable: VARIABLES.CAN_SENSOR_1 [0]
        Rectangle (207,36 25x24), "%2x", text variable: VARIABLES.CAN_SENSOR_1 [1]
        Rectangle (246,36 25x24), "%2x", text variable: VARIABLES.CAN_SENSOR_1 [2]
        Rectangle (275,36 25x24), "%2x", text variable: VARIABLES.CAN_SENSOR_1 [3]
        Rectangle (314,36 25x24), "%2x", text variable: VARIABLES.CAN_SENSOR_1 [4]
        Rectangle (343,36 25x24), "%2x", text variable: VARIABLES.CAN_SENSOR_1 [5]
        Rectangle (382,36 25x24), "%2x", text variable: VARIABLES.CAN_SENSOR_1 [6]
        Rectangle (411,36 25x24), "%2x", text variable: VARIABLES.CAN_SENSOR_1 [7]
        Rectangle (178,67 25x24), "%2x", text variable: VARIABLES.CAN_SENSOR_2 [0]
        Rectangle (207,67 25x24), "%2x", text variable: VARIABLES.CAN_SENSOR_2 [1]
        Rectangle (246,67 25x24), "%2x", text variable: VARIABLES.CAN_SENSOR_2 [2]
        Rectangle (275,67 25x24), "%2x", text variable: VARIABLES.CAN_SENSOR_2 [3]
        Rectangle (314,67 25x24), "%2x", text variable: VARIABLES.CAN_SENSOR_2 [4]
        Rectangle (343,67 25x24), "%2x", text variable: VARIABLES.CAN_SENSOR_2 [5]
        Rectangle (382,67 25x24), "%2x", text variable: VARIABLES.CAN_SENSOR_2 [6]
        Rectangle (411,67 25x24), "%2x", text variable: VARIABLES.CAN_SENSOR_2 [7]
        Rectangle (178,98 25x24), "%2x", text variable: VARIABLES.CAN_SENSOR_3 [0]
        Rectangle (207,98 25x24), "%2x", text variable: VARIABLES.CAN_SENSOR_3 [1]
        Rectangle (246,98 25x24), "%2x", text variable: VARIABLES.CAN_SENSOR_3 [2]
        Rectangle (275,98 25x24), "%2x", text variable: VARIABLES.CAN_SENSOR_3 [3]
        Rectangle (314,98 25x24), "%2x", text variable: VARIABLES.CAN_SENSOR_3 [4]
        Rectangle (343,98 25x24), "%2x", text variable: VARIABLES.CAN_SENSOR_3 [5]
        Rectangle (382,98 25x24), "%2x", text variable: VARIABLES.CAN_SENSOR_3 [6]
        Rectangle (411,98 25x24), "%2x", text variable: VARIABLES.CAN_SENSOR_3 [7]
        Rectangle (178,129 25x24), "%2x", text variable: VARIABLES.CAN_SENSOR_4 [0]
        Rectangle (207,129 25x24), "%2x", text variable: VARIABLES.CAN_SENSOR_4 [1]
        Rectangle (246,129 25x24), "%2x", text variable: VARIABLES.CAN_SENSOR_4 [2]
        Rectangle (275,129 25x24), "%2x", text variable: VARIABLES.CAN_SENSOR_4 [3]
        Rectangle (314,129 25x24), "%2x", text variable: VARIABLES.CAN_SENSOR_4 [4]
        Rectangle (343,129 25x24), "%2x", text variable: VARIABLES.CAN_SENSOR_4 [5]
        Rectangle (382,129 25x24), "%2x", text variable: VARIABLES.CAN_SENSOR_4 [6]
        Rectangle (411,129 25x24), "%2x", text variable: VARIABLES.CAN_SENSOR_4 [7]
        Rectangle (178,160 25x24), "%2x", text variable: VARIABLES.CAN_SENSOR_5 [0]
        Rectangle (207,160 25x24), "%2x", text variable: VARIABLES.CAN_SENSOR_5 [1]
        Rectangle (246,160 25x24), "%2x", text variable: VARIABLES.CAN_SENSOR_5 [2]
        Rectangle (275,160 25x24), "%2x", text variable: VARIABLES.CAN_SENSOR_5 [3]
        Rectangle (314,160 25x24), "%2x", text variable: VARIABLES.CAN_SENSOR_5 [4]
        Rectangle (343,160 25x24), "%2x", text variable: VARIABLES.CAN_SENSOR_5 [5]
        Rectangle (382,160 25x24), "%2x", text variable: VARIABLES.CAN_SENSOR_5 [6]
        Rectangle (411,160 25x24), "%2x", text variable: VARIABLES.CAN_SENSOR_5 [7]
        Rectangle (178,191 25x24), "%2x", text variable: VARIABLES.CAN_SENSOR_6[0]
        Rectangle (207,191 25x24), "%2x", text variable: VARIABLES.CAN_SENSOR_6[1]
        Rectangle (246,191 24x24), "%2x", text variable: VARIABLES.CAN_SENSOR_6 [2]
        Rectangle (275,191 25x24), "%2x", text variable: VARIABLES.CAN_SENSOR_6 [3]
        Rectangle (314,191 25x24), "%2x", text variable: VARIABLES.CAN_SENSOR_6[4]
        Rectangle (343,191 25x24), "%2x", text variable: VARIABLES.CAN_SENSOR_6 [5]
        Rectangle (382,191 25x24), "%2x", text variable: VARIABLES.CAN_SENSOR_6 [6]
        Rectangle (411,191 25x24), "%2x", text variable: VARIABLES.CAN_SENSOR_6[7]
        Rectangle (178,222 25x24), "%2x", text variable: VARIABLES.CAN_SENSOR_7 [0]
        Rectangle (207,222 25x24), "%2x", text variable: VARIABLES.CAN_SENSOR_7[1]
        Rectangle (246,222 25x24), "%2x", text variable: VARIABLES.CAN_SENSOR_7 [2]
        Rectangle (275,222 25x24), "%2x", text variable: VARIABLES.CAN_SENSOR_7 [3]
        Rectangle (314,222 25x24), "%2x", text variable: VARIABLES.CAN_SENSOR_7 [4]
        Rectangle (343,222 25x24), "%2x", text variable: VARIABLES.CAN_SENSOR_7 [5]
        Rectangle (382,222 25x24), "%2x", text variable: VARIABLES.CAN_SENSOR_7 [6]
        Rectangle (411,222 25x24), "%2x", text variable: VARIABLES.CAN_SENSOR_7 [7]
        Rectangle (135,36 24x24), "01"
        Rectangle (135,67 25x24), "02"
        Rectangle (135,98 25x24), "03"
        Rectangle (135,129 25x24), "04"
        Rectangle (135,160 25x24), "05"
        Rectangle (135,191 25x24), "1"
        Rectangle (135,191 25x24), "06"
        Rectangle (135,222 25x24), "07"
        Rectangle (178,253 25x24), "%2x", text variable: VARIABLES.CAN_SENSOR_8 [0]
        Rectangle (207,253 25x24), "%2x", text variable: VARIABLES.CAN_SENSOR_8[1]
        Rectangle (246,253 25x24), "%2x", text variable: VARIABLES.CAN_SENSOR_8 [2]
        Rectangle (275,253 25x24), "%2x", text variable: VARIABLES.CAN_SENSOR_8[3]
        Rectangle (314,253 25x24), "%2x", text variable: VARIABLES.CAN_SENSOR_8[4]
        Rectangle (343,253 25x24), "%2x", text variable: VARIABLES.CAN_SENSOR_8 [5]
        Rectangle (382,253 25x24), "%2x", text variable: VARIABLES.CAN_SENSOR_8 [6]
        Rectangle (411,253 25x24), "%2x", text variable: VARIABLES.CAN_SENSOR_8[7]
        Rectangle (178,284 25x24), "%2x", text variable: VARIABLES.CAN_SENSOR_9 [0]
        Rectangle (207,284 25x24), "%2x", text variable: VARIABLES.CAN_SENSOR_9 [1]
        Rectangle (246,284 25x24), "%2x", text variable: VARIABLES.CAN_SENSOR_9 [2]
        Rectangle (275,284 25x24), "%2x", text variable: VARIABLES.CAN_SENSOR_9 [3]
        Rectangle (314,284 25x24), "%2x", text variable: VARIABLES.CAN_SENSOR_9 [4]
        Rectangle (343,284 25x24), "%2x", text variable: VARIABLES.CAN_SENSOR_9 [5]
        Rectangle (382,284 25x24), "%2x", text variable: VARIABLES.CAN_SENSOR_9 [6]
        Rectangle (411,284 25x24), "%2x", text variable: VARIABLES.CAN_SENSOR_9 [7]
        Rectangle (178,315 25x24), "%2x", text variable: VARIABLES.CAN_SENSOR_10[0]
        Rectangle (207,315 25x24), "%2x", text variable: VARIABLES.CAN_SENSOR_10[1]
        Rectangle (246,315 25x24), "%2x", text variable: VARIABLES.CAN_SENSOR_10[2]
        Rectangle (275,315 25x24), "%2x", text variable: VARIABLES.CAN_SENSOR_10[3]
        Rectangle (314,315 25x24), "%2x", text variable: VARIABLES.CAN_SENSOR_10[4]
        Rectangle (343,315 25x24), "%2x", text variable: VARIABLES.CAN_SENSOR_10[5]
        Rectangle (382,315 25x24), "%2x", text variable: VARIABLES.CAN_SENSOR_10[6]
        Rectangle (411,315 25x24), "%2x", text variable: VARIABLES.CAN_SENSOR_10[7]
        Rectangle (135,253 25x24), "08"
        Rectangle (135,284 25x24), "1"
        Rectangle (135,284 25x24), "09"
        Rectangle (135,315 25x24), "10"
    Rectangle (968,11 117x15), "Sensor Positions"
    Image (892,47 305x305), image: PICTURES.1
    Line (41,9) (1191,9)
    Line (41,361) (1191,361)
    Line (481,380) (1191,380)
    Line (41,41) (1191,41)
END_VISUALIZATION

// ---- VISUs/VISUALISATION_STIFFNESS_COLLISION.TcVIS
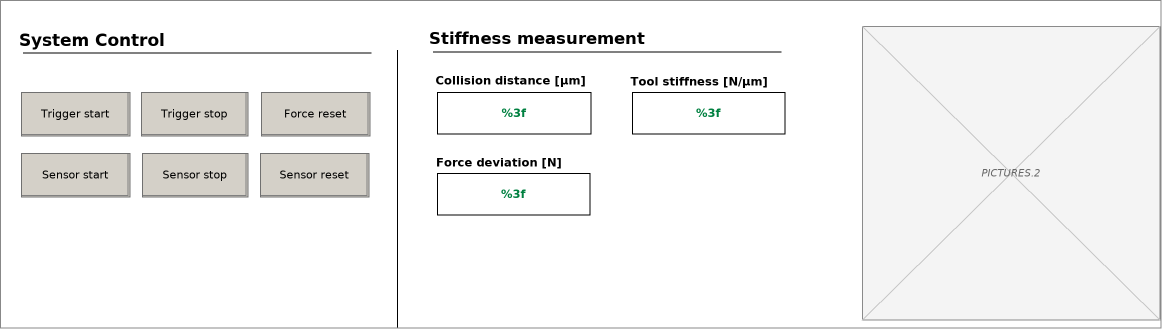
VISUALIZATION VISUALISATION_STIFFNESS_COLLISION  // 1162x329
    Button (21,92 109x44), "Trigger start"
        OnMouseClick: execute { VARIABLES.CAN_TRIGGER_STATE:=1; }
    Button (141,92 107x44), "Trigger stop"
        OnMouseClick: execute { VARIABLES.CAN_TRIGGER_STATE:=0; }
    Button (21,153 109x44), "Sensor start"
        OnMouseClick: execute { CAN_CONTROL_STATE:=1; }
    Button (142,153 106x44), "Sensor stop"
        OnMouseClick: execute { CAN_CONTROL_STATE:=0; }
    Button (260,153 109x44), "Sensor reset"
        OnMouseClick: execute { CAN_CONTROL_STATE:=2; }
    Button (261,92 109x44), "Force reset"
        OnMouseClick: execute { VARIABLES.FORCE_RESET:=1; }
    Rectangle (17,25 150x30), "System Control"
    Line (371,53) (23,53)
    Rectangle (428,31 218x15), "Stiffness measurement"
    Rectangle (632,92 153x42), "%3f", text variable: VARIABLES.TOOL_STIFFNESS_SELC_PTS[1,3]
    Rectangle (437,92 154x42), "%3f", text variable: VARIABLES.COLLISION_DISTANCE
    Rectangle (437,173 153x42), "%3f", text variable: VARIABLES.FORCE_DEVIATION[1]
    Rectangle (437,73 148x15), "Collision distance [µm]"
    Rectangle (437,155 124x15), "Force deviation [N]"
    Rectangle (632,74 135x15), "Tool stiffness [N/µm]"
    Line (397,50) (397,327)
    Line (781,52) (433,52)
    Image (862,26 298x294), image: PICTURES.2
END_VISUALIZATION
